C01828=1149.288,-103.464,-43.595,178.756,5.963,149.436
C01829=1149.282,-103.213,-43.605,178.759,5.964,149.436
C01830=1149.276,-102.942,-43.615,178.761,5.964,149.435
C01831=1149.271,-102.669,-43.625,178.763,5.965,149.435
C01832=1149.265,-102.397,-43.635,178.765,5.965,149.434
C01833=1149.260,-102.125,-43.645,178.767,5.965,149.433
C01834=1149.254,-101.875,-43.654,178.770,5.966,149.433
C01835=1149.249,-101.625,-43.664,178.772,5.966,149.432
C01836=1149.243,-101.375,-43.672,178.774,5.967,149.432
C01837=1149.238,-101.125,-43.681,178.775,5.966,149.431
C01838=1149.233,-100.877,-43.691,178.778,5.967,149.431
C01839=1149.227,-100.627,-43.700,178.780,5.968,149.430
C01840=1149.222,-100.377,-43.709,178.782,5.968,149.430
C01841=1149.216,-100.127,-43.718,178.784,5.968,149.429
C01842=1149.211,-99.877,-43.727,178.786,5.969,149.429
C01843=1149.206,-99.628,-43.737,178.788,5.969,149.428
C01844=1149.201,-99.378,-43.746,178.791,5.969,149.427
C01845=1149.195,-99.128,-43.755,178.792,5.969,149.427
C01846=1149.189,-98.878,-43.764,178.794,5.970,149.426
C01847=1149.185,-98.629,-43.774,178.797,5.971,149.426
C01848=1149.179,-98.378,-43.783,178.799,5.970,149.425
C01849=1149.174,-98.129,-43.792,178.801,5.971,149.425
C01850=1149.169,-97.879,-43.802,178.803,5.972,149.424
C01851=1149.163,-97.629,-43.811,178.805,5.972,149.424
C01852=1149.158,-97.379,-43.820,178.807,5.973,149.423
C01853=1149.152,-97.129,-43.829,178.809,5.972,149.423
C01854=1149.147,-96.880,-43.839,178.811,5.973,149.422
C01855=1149.142,-96.630,-43.848,178.813,5.974,149.422
C01856=1149.136,-96.380,-43.858,178.815,5.974,149.421
C01857=1149.131,-96.131,-43.867,178.818,5.974,149.420
C01858=1149.126,-95.881,-43.876,178.820,5.975,149.420
C01859=1149.120,-95.631,-43.886,178.821,5.975,149.419
C01860=1149.115,-95.381,-43.895,178.824,5.976,149.419
C01861=1149.109,-95.131,-43.905,178.826,5.975,149.418
C01862=1149.104,-94.882,-43.914,178.828,5.976,149.418
C01863=1149.099,-94.632,-43.923,178.830,5.977,149.417
C01864=1149.093,-94.382,-43.933,178.832,5.977,149.417
C01865=1149.088,-94.133,-43.942,178.834,5.977,149.416
C01866=1149.082,-93.883,-43.952,178.836,5.978,149.416
C01867=1149.077,-93.633,-43.961,178.838,5.978,149.415
C01868=1149.072,-93.384,-43.970,178.840,5.979,149.415
C01869=1149.066,-93.133,-43.980,178.843,5.979,149.414
C01870=1149.062,-92.884,-43.990,178.845,5.979,149.413
C01871=1149.056,-92.634,-43.999,178.847,5.980,149.413
C01872=1149.051,-92.384,-44.009,178.849,5.980,149.412
C01873=1149.046,-92.134,-44.019,178.851,5.980,149.412
C01874=1149.040,-91.884,-44.027,178.853,5.981,149.411
C01875=1149.035,-91.634,-44.038,178.855,5.982,149.411
C01876=1149.030,-91.385,-44.047,178.857,5.982,149.410
C01877=1149.024,-91.135,-44.057,178.860,5.982,149.410
C01878=1149.019,-90.885,-44.066,178.862,5.983,149.409
C01879=1149.013,-90.636,-44.076,178.863,5.983,149.409
C01880=1149.008,-90.386,-44.085,178.866,5.983,149.408
C01881=1149.003,-90.137,-44.094,178.868,5.984,149.407
C01882=1148.997,-89.886,-44.104,178.870,5.984,149.407
C01883=1148.992,-89.637,-44.113,178.872,5.985,149.406
C01884=1148.987,-89.387,-44.123,178.874,5.984,149.406
C01885=1148.982,-89.137,-44.133,178.876,5.985,149.405
C01886=1148.976,-88.887,-44.142,178.879,5.986,149.405
C01887=1148.971,-88.637,-44.153,178.881,5.986,149.404
C01888=1148.966,-88.388,-44.162,178.883,5.986,149.404
C01889=1148.960,-88.138,-44.172,178.885,5.987,149.403
C01890=1148.955,-87.889,-44.181,178.887,5.987,149.403
C01891=1148.949,-87.639,-44.191,178.889,5.987,149.402
C01892=1148.944,-87.389,-44.200,178.891,5.988,149.401
C01893=1148.939,-87.138,-44.210,178.894,5.989,149.401
C01894=1148.934,-86.889,-44.220,178.895,5.989,149.400
C01895=1148.929,-86.640,-44.230,178.897,5.989,149.400
C01896=1148.923,-86.390,-44.239,178.900,5.990,149.399
C01897=1148.918,-86.140,-44.249,178.902,5.990,149.399
C01898=1148.912,-85.890,-44.259,178.904,5.990,149.398
C01899=1148.907,-85.641,-44.268,178.907,5.991,149.398
C01900=1148.902,-85.391,-44.279,178.908,5.991,149.397
C01901=1148.897,-85.141,-44.288,178.910,5.992,149.397
C01902=1148.891,-84.891,-44.298,178.913,5.992,149.396
C01903=1148.886,-84.642,-44.308,178.915,5.992,149.395
C01904=1148.881,-84.392,-44.317,178.917,5.993,149.395
C01905=1148.875,-84.142,-44.327,178.919,5.993,149.394
C01906=1148.871,-83.892,-44.337,178.921,5.993,149.394
C01907=1148.865,-83.642,-44.347,178.923,5.994,149.393
C01908=1148.859,-83.393,-44.357,178.925,5.995,149.393
C01909=1148.854,-83.143,-44.367,178.928,5.995,149.392
C01910=1148.848,-82.893,-44.376,178.930,5.995,149.392
C01911=1148.844,-82.643,-44.386,178.932,5.996,149.391
C01912=1148.839,-82.394,-44.396,178.934,5.996,149.391
C01913=1148.833,-82.144,-44.406,178.936,5.996,149.390
C01914=1148.828,-81.894,-44.415,178.938,5.997,149.389
C01915=1148.822,-81.645,-44.426,178.941,5.998,149.389
C01916=1148.817,-81.395,-44.436,178.943,5.997,149.388
C01917=1148.812,-81.145,-44.445,178.945,5.998,149.388
C01918=1148.806,-80.895,-44.455,178.947,5.999,149.387
C01919=1148.801,-80.646,-44.466,178.949,5.999,149.387
C01920=1148.796,-80.396,-44.475,178.951,5.999,149.386
C01921=1148.791,-80.146,-44.485,178.954,6.000,149.386
C01922=1148.785,-79.896,-44.495,178.956,6.001,149.385
C01923=1148.779,-79.647,-44.505,178.958,6.000,149.384
C01924=1148.775,-79.397,-44.515,178.960,6.001,149.384
C01925=1148.770,-79.147,-44.526,178.962,6.002,149.383
C01926=1148.764,-78.897,-44.535,178.965,6.002,149.383
C01927=1148.759,-78.648,-44.545,178.966,6.002,149.382
C01928=1148.753,-78.398,-44.555,178.969,6.003,149.382
C01929=1148.748,-78.149,-44.565,178.971,6.003,149.381
C01930=1148.743,-77.898,-44.576,178.973,6.003,149.381
C01931=1148.738,-77.648,-44.585,178.975,6.004,149.380
C01932=1148.732,-77.399,-44.595,178.977,6.005,149.380
C01933=1148.726,-77.149,-44.605,178.980,6.005,149.379
C01934=1148.721,-76.878,-44.616,178.982,6.006,149.378
C01935=1148.715,-76.606,-44.628,178.984,6.005,149.378
C01936=1148.710,-76.335,-44.638,178.986,6.006,149.377
C01937=1148.703,-76.064,-44.649,178.989,6.007,149.377
C01938=1148.698,-75.813,-44.660,178.991,6.007,149.376
C01939=1148.693,-75.564,-44.669,178.993,6.008,149.376
C01940=1148.688,-75.315,-44.679,178.996,6.008,149.375
C01941=1148.682,-75.065,-44.690,178.998,6.008,149.374
C01942=1148.677,-74.815,-44.700,179.000,6.009,149.374
C01943=1148.672,-74.565,-44.710,179.003,6.010,149.373
C01944=1148.667,-74.316,-44.720,179.004,6.010,149.373
C01945=1148.662,-74.066,-44.731,179.006,6.010,149.372
C01946=1148.656,-73.816,-44.741,179.009,6.011,149.372
C01947=1148.650,-73.567,-44.751,179.011,6.012,149.371
C01948=1148.645,-73.317,-44.761,179.013,6.012,149.371
C01949=1148.640,-73.066,-44.771,179.016,6.012,149.370
C01950=1148.634,-72.817,-44.781,179.018,6.013,149.369
C01951=1148.629,-72.568,-44.791,179.020,6.013,149.369
C01952=1148.624,-72.317,-44.801,179.022,6.013,149.368
C01953=1148.619,-72.068,-44.812,179.024,6.014,149.368
C01954=1148.613,-71.818,-44.822,179.026,6.015,149.367
C01955=1148.608,-71.568,-44.832,179.029,6.015,149.366
C01956=1148.602,-71.318,-44.843,179.031,6.015,149.366
C01957=1148.597,-71.069,-44.853,179.033,6.016,149.366
C01958=1148.593,-70.820,-44.863,179.035,6.016,149.365
C01959=1148.587,-70.570,-44.874,179.038,6.017,149.364
C01960=1148.582,-70.321,-44.884,179.039,6.017,149.364
C01961=1148.577,-70.070,-44.894,179.042,6.017,149.363
C01962=1148.571,-69.821,-44.905,179.044,6.018,149.363
C01963=1148.566,-69.570,-44.915,179.046,6.019,149.362
C01964=1148.560,-69.321,-44.925,179.048,6.018,149.361
C01965=1148.555,-69.071,-44.936,179.051,6.019,149.361
C01966=1148.550,-68.821,-44.946,179.053,6.020,149.361
C01967=1148.544,-68.572,-44.956,179.055,6.020,149.360
C01968=1148.539,-68.322,-44.967,179.057,6.020,149.359
C01969=1148.534,-68.072,-44.977,179.059,6.021,149.359
C01970=1148.528,-67.822,-44.987,179.062,6.021,149.358
C01971=1148.524,-67.573,-44.998,179.064,6.022,149.358
C01972=1148.518,-67.323,-45.008,179.066,6.023,149.357
C01973=1148.513,-67.074,-45.019,179.068,6.023,149.356
C01974=1148.508,-66.824,-45.029,179.071,6.023,149.356
C01975=1148.502,-66.574,-45.039,179.073,6.024,149.355
C01976=1148.497,-66.324,-45.050,179.075,6.025,149.355
C01977=1148.492,-66.075,-45.061,179.077,6.024,149.354
C01978=1148.486,-65.825,-45.071,179.080,6.025,149.354
C01979=1148.481,-65.575,-45.082,179.082,6.026,149.353
C01980=1148.476,-65.326,-45.092,179.084,6.026,149.353
C01981=1148.471,-65.075,-45.102,179.087,6.027,149.352
C01982=1148.465,-64.826,-45.113,179.088,6.027,149.351
C01983=1148.460,-64.576,-45.124,179.090,6.028,149.351
C01984=1148.455,-64.327,-45.134,179.093,6.028,149.350
C01985=1148.450,-64.076,-45.145,179.095,6.029,149.350
C01986=1148.444,-63.827,-45.155,179.098,6.030,149.349
C01987=1148.439,-63.578,-45.166,179.100,6.029,149.349
C01988=1148.434,-63.328,-45.176,179.102,6.030,149.348
C01989=1148.428,-63.078,-45.187,179.104,6.031,149.348
C01990=1148.423,-62.828,-45.197,179.107,6.031,149.347
C01991=1148.417,-62.579,-45.209,179.109,6.032,149.346
C01992=1148.412,-62.328,-45.219,179.111,6.031,149.346
C01993=1148.407,-62.079,-45.229,179.113,6.032,149.345
C01994=1148.402,-61.829,-45.241,179.115,6.033,149.345
C01995=1148.396,-61.580,-45.251,179.118,6.033,149.344
C01996=1148.391,-61.329,-45.262,179.120,6.034,149.344
C01997=1148.386,-61.081,-45.272,179.122,6.034,149.343
C01998=1148.381,-60.830,-45.283,179.124,6.035,149.342
C01999=1148.376,-60.581,-45.293,179.127,6.035,149.342
C02000=1148.371,-60.331,-45.305,179.129,6.036,149.341
C02001=1148.365,-60.082,-45.315,179.131,6.036,149.341
C02002=1148.360,-59.831,-45.325,179.133,6.036,149.340
C02003=1148.354,-59.582,-45.337,179.136,6.037,149.340
C02004=1148.349,-59.332,-45.347,179.138,6.038,149.339
C02005=1148.344,-59.082,-45.358,179.140,6.038,149.339
C02006=1148.339,-58.833,-45.369,179.143,6.039,149.338
C02007=1148.333,-58.583,-45.379,179.145,6.040,149.337
C02008=1148.329,-58.334,-45.390,179.147,6.040,149.337
C02009=1148.323,-58.084,-45.401,179.149,6.040,149.336
C02010=1148.318,-57.834,-45.411,179.151,6.041,149.336
C02011=1148.313,-57.584,-45.423,179.154,6.041,149.335
C02012=1148.307,-57.334,-45.433,179.156,6.042,149.335
C02013=1148.302,-57.085,-45.445,179.158,6.042,149.334
C02014=1148.297,-56.835,-45.455,179.161,6.042,149.333
C02015=1148.292,-56.585,-45.466,179.163,6.043,149.333
C02016=1148.287,-56.336,-45.476,179.165,6.044,149.332
C02017=1148.281,-56.085,-45.487,179.168,6.044,149.332
C02018=1148.275,-55.836,-45.498,179.170,6.045,149.331
C02019=1148.270,-55.586,-45.509,179.172,6.045,149.331
C02020=1148.266,-55.337,-45.520,179.174,6.045,149.330
C02021=1148.260,-55.087,-45.530,179.176,6.046,149.330
C02022=1148.255,-54.837,-45.542,179.179,6.047,149.329
C02023=1148.249,-54.588,-45.553,179.181,6.047,149.328
C02024=1148.244,-54.338,-45.564,179.183,6.048,149.328
C02025=1148.240,-54.088,-45.575,179.186,6.049,149.327
C02026=1148.234,-53.839,-45.585,179.188,6.049,149.327
C02027=1148.229,-53.589,-45.597,179.190,6.049,149.326
C02028=1148.223,-53.339,-45.607,179.192,6.050,149.326
C02029=1148.218,-53.090,-45.619,179.195,6.050,149.325
C02030=1148.213,-52.839,-45.629,179.197,6.051,149.324
C02031=1148.207,-52.590,-45.641,179.199,6.052,149.324
C02032=1148.202,-52.340,-45.651,179.202,6.052,149.323
C02033=1148.197,-52.091,-45.662,179.204,6.052,149.323
C02034=1148.192,-51.841,-45.674,179.206,6.053,149.322
C02035=1148.187,-51.591,-45.685,179.209,6.053,149.322
C02036=1148.181,-51.342,-45.696,179.211,6.054,149.321
C02037=1148.176,-51.092,-45.706,179.213,6.055,149.321
C02038=1148.171,-50.821,-45.719,179.216,6.055,149.320
C02039=1148.165,-50.550,-45.730,179.218,6.056,149.319
C02040=1148.159,-50.279,-45.743,179.220,6.056,149.319
C02041=1148.153,-50.009,-45.755,179.223,6.057,149.318
C02042=1148.148,-49.759,-45.766,179.225,6.058,149.318
C02043=1148.143,-49.510,-45.777,179.228,6.058,149.317
C02044=1148.137,-49.260,-45.788,179.230,6.059,149.316
C02045=1148.132,-49.010,-45.799,179.232,6.059,149.316
C02046=1148.128,-48.761,-45.811,179.234,6.059,149.315
C02047=1148.121,-48.511,-45.821,179.237,6.060,149.315
C02048=1148.117,-48.261,-45.833,179.239,6.060,149.314
C02049=1148.112,-48.012,-45.844,179.241,6.061,149.314
C02050=1148.106,-47.762,-45.855,179.244,6.062,149.313
C02051=1148.101,-47.512,-45.866,179.246,6.062,149.312
C02052=1148.095,-47.262,-45.878,179.249,6.063,149.312
C02053=1148.091,-47.013,-45.889,179.251,6.063,149.311
C02054=1148.085,-46.764,-45.900,179.253,6.063,149.311
C02055=1148.080,-46.513,-45.911,179.255,6.064,149.310
C02056=1148.075,-46.263,-45.923,179.258,6.065,149.310
C02057=1148.069,-46.014,-45.934,179.260,6.065,149.309
C02058=1148.064,-45.765,-45.945,179.262,6.066,149.308
C02059=1148.059,-45.514,-45.956,179.265,6.067,149.308
C02060=1148.053,-45.265,-45.967,179.267,6.067,149.307
C02061=1148.049,-45.016,-45.979,179.270,6.068,149.307
C02062=1148.043,-44.766,-45.991,179.271,6.068,149.306
C02063=1148.038,-44.516,-46.002,179.274,6.068,149.305
C02064=1148.032,-44.266,-46.013,179.276,6.069,149.305
C02065=1148.027,-44.016,-46.024,179.278,6.070,149.305
C02066=1148.022,-43.767,-46.036,179.281,6.070,149.304
C02067=1148.017,-43.517,-46.047,179.283,6.071,149.303
C02068=1148.012,-43.268,-46.058,179.286,6.071,149.303
C02069=1148.007,-43.018,-46.070,179.288,6.072,149.302
C02070=1148.002,-42.768,-46.081,179.290,6.073,149.302
C02071=1147.996,-42.518,-46.092,179.293,6.073,149.301
C02072=1147.991,-42.269,-46.103,179.295,6.074,149.301
C02073=1147.985,-42.019,-46.115,179.297,6.074,149.300
C02074=1147.981,-41.769,-46.127,179.299,6.074,149.299
C02075=1147.975,-41.519,-46.138,179.301,6.075,149.299
C02076=1147.970,-41.271,-46.149,179.304,6.076,149.298
C02077=1147.965,-41.021,-46.161,179.306,6.076,149.298
C02078=1147.960,-40.771,-46.173,179.309,6.077,149.297
C02079=1147.955,-40.521,-46.184,179.311,6.078,149.297
C02080=1147.949,-40.271,-46.196,179.314,6.078,149.296
C02081=1147.944,-40.022,-46.207,179.316,6.079,149.295
C02082=1147.938,-39.772,-46.219,179.318,6.080,149.295
C02083=1147.934,-39.523,-46.230,179.321,6.080,149.294
C02084=1147.928,-39.272,-46.242,179.323,6.081,149.294
C02085=1147.923,-39.022,-46.253,179.325,6.080,149.293
C02086=1147.917,-38.773,-46.264,179.327,6.081,149.293
C02087=1147.913,-38.524,-46.276,179.329,6.082,149.292
C02088=1147.907,-38.274,-46.288,179.332,6.082,149.291
C02089=1147.902,-38.024,-46.299,179.334,6.083,149.291
C02090=1147.897,-37.774,-46.311,179.337,6.084,149.290
C02091=1147.892,-37.525,-46.323,179.339,6.084,149.290
C02092=1147.887,-37.276,-46.334,179.341,6.085,149.289
C02093=1147.881,-37.026,-46.346,179.344,6.086,149.289
C02094=1147.876,-36.776,-46.358,179.346,6.086,149.288
C02095=1147.871,-36.526,-46.369,179.349,6.087,149.287
C02096=1147.866,-36.276,-46.381,179.351,6.088,149.287
C02097=1147.860,-36.026,-46.393,179.354,6.088,149.286
C02098=1147.855,-35.778,-46.404,179.356,6.089,149.286
C02099=1147.849,-35.528,-46.416,179.358,6.090,149.285
C02100=1147.844,-35.278,-46.428,179.361,6.090,149.285
C02101=1147.839,-35.028,-46.439,179.363,6.091,149.284
C02102=1147.834,-34.778,-46.451,179.365,6.091,149.283
C02103=1147.829,-34.528,-46.462,179.367,6.091,149.283
C02104=1147.824,-34.279,-46.475,179.370,6.092,149.282
C02105=1147.819,-34.029,-46.487,179.372,6.092,149.282
C02106=1147.813,-33.780,-46.498,179.374,6.093,149.281
C02107=1147.808,-33.530,-46.510,179.377,6.094,149.281
C02108=1147.802,-33.280,-46.521,179.379,6.094,149.280
C02109=1147.797,-33.030,-46.533,179.382,6.095,149.279
C02110=1147.793,-32.781,-46.545,179.384,6.096,149.279
C02111=1147.787,-32.532,-46.557,179.386,6.096,149.278
C02112=1147.782,-32.282,-46.569,179.389,6.097,149.278
C02113=1147.777,-32.032,-46.580,179.391,6.098,149.277
C02114=1147.772,-31.782,-46.592,179.393,6.098,149.277
C02115=1147.767,-31.533,-46.605,179.396,6.099,149.276
C02116=1147.761,-31.283,-46.617,179.398,6.099,149.275
C02117=1147.756,-31.034,-46.628,179.401,6.100,149.275
C02118=1147.750,-30.784,-46.640,179.403,6.101,149.274
C02119=1147.745,-30.535,-46.652,179.405,6.101,149.274
C02120=1147.740,-30.285,-46.664,179.408,6.102,149.273
C02121=1147.735,-30.035,-46.675,179.410,6.102,149.273
C02122=1147.730,-29.785,-46.687,179.412,6.103,149.272
C02123=1147.725,-29.536,-46.700,179.415,6.104,149.271
C02124=1147.719,-29.286,-46.712,179.417,6.104,149.271
C02125=1147.714,-29.036,-46.723,179.419,6.105,149.270
C02126=1147.709,-28.787,-46.736,179.422,6.106,149.270
C02127=1147.704,-28.537,-46.748,179.424,6.106,149.269
C02128=1147.698,-28.287,-46.759,179.427,6.107,149.269
C02129=1147.693,-28.037,-46.771,179.429,6.108,149.268
C02130=1147.689,-27.788,-46.783,179.432,6.108,149.267
C02131=1147.683,-27.538,-46.795,179.434,6.109,149.267
C02132=1147.678,-27.289,-46.808,179.436,6.110,149.266
C02133=1147.673,-27.039,-46.820,179.439,6.110,149.266
C02134=1147.667,-26.789,-46.832,179.441,6.111,149.265
C02135=1147.662,-26.540,-46.844,179.444,6.111,149.265
C02136=1147.657,-26.290,-46.855,179.446,6.112,149.264
C02137=1147.652,-26.040,-46.867,179.448,6.112,149.263
C02138=1147.647,-25.791,-46.880,179.451,6.113,149.263
C02139=1147.641,-25.541,-46.892,179.453,6.114,149.262
C02140=1147.636,-25.292,-46.904,179.456,6.114,149.262
C02141=1147.631,-25.042,-46.916,179.458,6.115,149.261
C02142=1147.626,-24.771,-46.929,179.460,6.116,149.261
C02143=1147.620,-24.502,-46.943,179.463,6.116,149.260
C02144=1147.615,-24.232,-46.956,179.465,6.117,149.259
C02145=1147.609,-23.961,-46.969,179.468,6.118,149.259
C02146=1147.604,-23.712,-46.982,179.471,6.119,149.258
C02147=1147.599,-23.462,-46.993,179.473,6.119,149.258
C02148=1147.594,-23.213,-47.006,179.476,6.120,149.257
C02149=1147.588,-22.963,-47.017,179.478,6.121,149.256
C02150=1147.583,-22.714,-47.030,179.480,6.121,149.256
C02151=1147.578,-22.464,-47.042,179.483,6.122,149.255
C02152=1147.573,-22.214,-47.055,179.485,6.123,149.255
C02153=1147.567,-21.964,-47.066,179.487,6.123,149.254
C02154=1147.562,-21.715,-47.079,179.490,6.124,149.254
C02155=1147.557,-21.465,-47.091,179.492,6.125,149.253
C02156=1147.551,-21.216,-47.104,179.495,6.125,149.252
C02157=1147.546,-20.966,-47.115,179.497,6.126,149.252
C02158=1147.541,-20.717,-47.128,179.499,6.127,149.251
C02159=1147.536,-20.466,-47.140,179.502,6.127,149.251
C02160=1147.531,-20.217,-47.153,179.504,6.128,149.250
C02161=1147.526,-19.967,-47.165,179.507,6.128,149.250
C02162=1147.520,-19.717,-47.177,179.509,6.129,149.249
C02163=1147.515,-19.468,-47.190,179.512,6.129,149.248
C02164=1147.510,-19.218,-47.202,179.514,6.130,149.248
C02165=1147.505,-18.969,-47.214,179.516,6.131,149.247
C02166=1147.500,-18.720,-47.227,179.519,6.131,149.247
C02167=1147.494,-18.470,-47.239,179.521,6.132,149.246
C02168=1147.490,-18.220,-47.252,179.523,6.133,149.246
C02169=1147.485,-17.970,-47.264,179.526,6.133,149.245
C02170=1147.479,-17.720,-47.276,179.528,6.134,149.245
C02171=1147.474,-17.471,-47.289,179.531,6.135,149.244
C02172=1147.469,-17.222,-47.302,179.534,6.136,149.243
C02173=1147.463,-16.972,-47.313,179.536,6.137,149.243
C02174=1147.458,-16.722,-47.326,179.538,6.138,149.242
C02175=1147.453,-16.472,-47.340,179.541,6.138,149.242
C02176=1147.448,-16.222,-47.352,179.543,6.139,149.241
C02177=1147.443,-15.973,-47.364,179.546,6.139,149.241
C02178=1147.437,-15.724,-47.377,179.548,6.140,149.240
C02179=1147.432,-15.474,-47.389,179.550,6.140,149.239
C02180=1147.427,-15.224,-47.401,179.553,6.141,149.239
C02181=1147.422,-14.974,-47.414,179.555,6.142,149.238
C02182=1147.417,-14.725,-47.427,179.557,6.142,149.238
C02183=1147.412,-14.476,-47.439,179.560,6.143,149.237
C02184=1147.407,-14.226,-47.451,179.562,6.144,149.237
C02185=1147.401,-13.976,-47.464,179.564,6.144,149.236
C02186=1147.396,-13.726,-47.477,179.568,6.146,149.235
C02187=1147.391,-13.477,-47.490,179.570,6.146,149.235
C02188=1147.386,-13.227,-47.503,179.573,6.147,149.234
C02189=1147.381,-12.977,-47.515,179.575,6.148,149.234
C02190=1147.375,-12.728,-47.527,179.577,6.148,149.233
C02191=1147.370,-12.478,-47.541,179.580,6.149,149.233
C02192=1147.365,-12.229,-47.553,179.582,6.150,149.232
C02193=1147.360,-11.979,-47.566,179.584,6.150,149.231
C02194=1147.355,-11.730,-47.578,179.587,6.151,149.231
C02195=1147.350,-11.480,-47.591,179.589,6.151,149.230
C02196=1147.345,-11.230,-47.603,179.591,6.152,149.230
C02197=1147.339,-10.980,-47.617,179.595,6.153,149.229
C02198=1147.334,-10.731,-47.629,179.597,6.154,149.229
C02199=1147.329,-10.481,-47.642,179.599,6.155,149.228
C02200=1147.324,-10.232,-47.655,179.602,6.155,149.228
C02201=1147.319,-9.982,-47.667,179.604,6.156,149.227
C02202=1147.313,-9.733,-47.680,179.607,6.157,149.226
C02203=1147.309,-9.483,-47.693,179.609,6.157,149.226
C02204=1147.304,-9.233,-47.706,179.611,6.158,149.225
C02205=1147.298,-8.984,-47.719,179.614,6.159,149.225
C02206=1147.293,-8.734,-47.732,179.616,6.159,149.224
C02207=1147.288,-8.484,-47.745,179.619,6.161,149.224
C02208=1147.283,-8.235,-47.757,179.621,6.162,149.223
C02209=1147.278,-7.986,-47.770,179.624,6.162,149.222
C02210=1147.273,-7.735,-47.784,179.626,6.163,149.222
C02211=1147.267,-7.486,-47.796,179.629,6.163,149.221
C02212=1147.262,-7.237,-47.809,179.631,6.164,149.221
C02213=1147.257,-6.986,-47.822,179.633,6.164,149.220
C02214=1147.252,-6.737,-47.835,179.636,6.165,149.220
C02215=1147.247,-6.488,-47.848,179.638,6.166,149.219
C02216=1147.241,-6.238,-47.861,179.641,6.167,149.218
C02217=1147.236,-5.988,-47.874,179.643,6.168,149.218
C02218=1147.231,-5.739,-47.886,179.646,6.169,149.217
C02219=1147.225,-5.489,-47.899,179.648,6.169,149.217
C02220=1147.221,-5.239,-47.912,179.651,6.170,149.216
C02221=1147.216,-4.990,-47.925,179.653,6.171,149.216
C02222=1147.210,-4.740,-47.938,179.656,6.171,149.215
C02223=1147.205,-4.490,-47.951,179.658,6.173,149.215
C02224=1147.200,-4.241,-47.964,179.661,6.173,149.214
C02225=1147.195,-3.991,-47.978,179.663,6.174,149.213
C02226=1147.190,-3.742,-47.991,179.665,6.175,149.213
C02227=1147.185,-3.493,-48.003,179.668,6.175,149.212
C02228=1147.180,-3.242,-48.017,179.670,6.176,149.212
C02229=1147.175,-2.993,-48.029,179.673,6.176,149.211
C02230=1147.169,-2.743,-48.043,179.676,6.178,149.211
C02231=1147.165,-2.494,-48.056,179.678,6.178,149.210
C02232=1147.160,-2.245,-48.069,179.680,6.179,149.209
C02233=1147.154,-1.994,-48.083,179.683,6.180,149.209
C02234=1147.149,-1.745,-48.095,179.685,6.180,149.208
C02235=1147.143,-1.495,-48.108,179.687,6.181,149.208
C02236=1147.139,-1.246,-48.122,179.690,6.182,149.207
C02237=1147.133,-0.996,-48.135,179.693,6.183,149.207
C02238=1147.128,-0.747,-48.148,179.696,6.184,149.206
C02239=1147.123,-0.497,-48.161,179.698,6.185,149.206
C02240=1147.118,-0.247,-48.174,179.700,6.185,149.205
C02241=1147.113,0.002,-48.188,179.703,6.186,149.204
C02242=1147.108,0.252,-48.201,179.705,6.187,149.204
C02243=1147.103,0.502,-48.214,179.708,6.188,149.203
C02244=1147.098,0.751,-48.228,179.710,6.189,149.203
C02245=1147.092,1.000,-48.240,179.713,6.189,149.202
C02246=1147.087,1.270,-48.255,179.715,6.190,149.202
C02247=1147.081,1.539,-48.270,179.718,6.191,149.201
C02248=1147.075,1.810,-48.284,179.721,6.192,149.200
C02249=1147.070,2.078,-48.298,179.723,6.192,149.200
C02250=1147.065,2.328,-48.311,179.726,6.193,149.199
C02251=1147.060,2.577,-48.325,179.729,6.194,149.199
C02252=1147.055,2.827,-48.338,179.731,6.195,149.198
C02253=1147.050,3.077,-48.351,179.733,6.196,149.197
C02254=1147.045,3.326,-48.365,179.736,6.196,149.197
C02255=1147.040,3.576,-48.378,179.738,6.197,149.196
C02256=1147.034,3.826,-48.391,179.741,6.199,149.196
C02257=1147.029,4.075,-48.405,179.744,6.199,149.195
C02258=1147.024,4.325,-48.418,179.746,6.200,149.195
C02259=1147.019,4.574,-48.432,179.748,6.200,149.194
C02260=1147.014,4.824,-48.445,179.751,6.201,149.194
C02261=1147.008,5.074,-48.458,179.754,6.202,149.193
C02262=1147.003,5.323,-48.473,179.756,6.203,149.192
C02263=1146.998,5.573,-48.485,179.759,6.203,149.192
C02264=1146.993,5.822,-48.499,179.761,6.204,149.191
C02265=1146.988,6.072,-48.512,179.763,6.205,149.191
C02266=1146.983,6.321,-48.526,179.766,6.206,149.190
C02267=1146.977,6.571,-48.540,179.768,6.207,149.190
C02268=1146.973,6.820,-48.553,179.771,6.208,149.189
C02269=1146.967,7.070,-48.566,179.773,6.208,149.188
C02270=1146.963,7.319,-48.580,179.776,6.209,149.188
C02271=1146.957,7.569,-48.593,179.779,6.210,149.187
C02272=1146.952,7.819,-48.608,179.781,6.211,149.187
C02273=1146.947,8.068,-48.620,179.784,6.212,149.186
C02274=1146.942,8.318,-48.634,179.786,6.213,149.186
C02275=1146.937,8.568,-48.648,179.788,6.213,149.185
C02276=1146.932,8.817,-48.661,179.791,6.215,149.185
C02277=1146.927,9.067,-48.676,179.794,6.215,149.184
C02278=1146.921,9.316,-48.689,179.796,6.216,149.183
C02279=1146.916,9.566,-48.703,179.799,6.216,149.183
C02280=1146.911,9.815,-48.716,179.801,6.218,149.182
C02281=1146.906,10.065,-48.730,179.804,6.219,149.182
C02282=1146.901,10.315,-48.744,179.806,6.219,149.181
C02283=1146.896,10.564,-48.757,179.808,6.220,149.181
C02284=1146.891,10.814,-48.771,179.811,6.220,149.180
C02285=1146.885,11.063,-48.784,179.814,6.222,149.180
C02286=1146.880,11.313,-48.799,179.816,6.223,149.179
C02287=1146.876,11.562,-48.812,179.819,6.223,149.178
C02288=1146.870,11.812,-48.825,179.821,6.224,149.178
C02289=1146.865,12.062,-48.840,179.824,6.225,149.177
C02290=1146.860,12.311,-48.854,179.826,6.226,149.177
C02291=1146.856,12.560,-48.867,179.829,6.227,149.176
C02292=1146.850,12.810,-48.881,179.831,6.227,149.176
C02293=1146.845,13.059,-48.895,179.834,6.229,149.175
C02294=1146.840,13.309,-48.909,179.836,6.230,149.174
C02295=1146.835,13.560,-48.923,179.839,6.230,149.174
C02296=1146.830,13.808,-48.936,179.841,6.231,149.173
C02297=1146.825,14.058,-48.950,179.844,6.232,149.173
C02298=1146.820,14.308,-48.965,179.847,6.233,149.172
C02299=1146.814,14.557,-48.978,179.849,6.234,149.172
C02300=1146.809,14.807,-48.992,179.852,6.234,149.171
C02301=1146.804,15.057,-49.006,179.854,6.236,149.171
C02302=1146.799,15.305,-49.020,179.857,6.236,149.170
C02303=1146.794,15.555,-49.034,179.859,6.237,149.169
C02304=1146.789,15.805,-49.047,179.861,6.238,149.169
C02305=1146.784,16.054,-49.061,179.865,6.239,149.168
C02306=1146.779,16.304,-49.076,179.867,6.240,149.168
C02307=1146.774,16.554,-49.090,179.869,6.240,149.167
C02308=1146.768,16.803,-49.104,179.872,6.242,149.167
C02309=1146.763,17.053,-49.118,179.875,6.242,149.166
C02310=1146.759,17.303,-49.131,179.877,6.243,149.166
C02311=1146.753,17.552,-49.145,179.879,6.244,149.165
C02312=1146.748,17.801,-49.159,179.882,6.245,149.164
C02313=1146.743,18.051,-49.174,179.885,6.246,149.164
C02314=1146.738,18.301,-49.188,179.887,6.247,149.163
C02315=1146.733,18.550,-49.202,179.889,6.247,149.163
C02316=1146.728,18.799,-49.216,179.893,6.249,149.162
C02317=1146.723,19.049,-49.230,179.895,6.249,149.162
C02318=1146.718,19.299,-49.245,179.897,6.250,149.161
C02319=1146.712,19.548,-49.258,179.900,6.252,149.161
C02320=1146.707,19.798,-49.273,179.902,6.252,149.160
C02321=1146.702,20.047,-49.287,179.905,6.253,149.159
C02322=1146.697,20.298,-49.301,179.908,6.254,149.159
C02323=1146.691,20.547,-49.314,179.910,6.255,149.158
C02324=1146.686,20.796,-49.329,179.913,6.256,149.158
C02325=1146.682,21.046,-49.343,179.915,6.257,149.157
C02326=1146.677,21.296,-49.357,179.918,6.258,149.157
C02327=1146.671,21.545,-49.371,179.920,6.259,149.156
C02328=1146.666,21.794,-49.386,179.923,6.259,149.156
C02329=1146.661,22.044,-49.400,179.926,6.261,149.155
C02330=1146.656,22.293,-49.415,179.928,6.261,149.154
C02331=1146.652,22.543,-49.429,179.930,6.262,149.154
C02332=1146.646,22.792,-49.443,179.933,6.264,149.154
C02333=1146.641,23.042,-49.457,179.936,6.264,149.153
C02334=1146.636,23.291,-49.471,179.938,6.265,149.152
C02335=1146.631,23.541,-49.486,179.941,6.265,149.152
C02336=1146.626,23.791,-49.500,179.943,6.267,149.151
C02337=1146.621,24.040,-49.514,179.946,6.267,149.151
C02338=1146.616,24.290,-49.528,179.948,6.268,149.150
C02339=1146.611,24.539,-49.543,179.951,6.270,149.150
C02340=1146.606,24.788,-49.558,179.954,6.270,149.149
C02341=1146.601,25.038,-49.572,179.956,6.271,149.149
C02342=1146.596,25.288,-49.586,179.959,6.272,149.148
C02343=1146.591,25.537,-49.600,179.961,6.273,149.147
C02344=1146.585,25.787,-49.615,179.963,6.274,149.147
C02345=1146.580,26.037,-49.629,179.967,6.275,149.146
C02346=1146.575,26.286,-49.644,179.969,6.276,149.146
C02347=1146.570,26.535,-49.658,179.971,6.277,149.145
C02348=1146.565,26.785,-49.673,179.974,6.278,149.145
C02349=1146.560,27.035,-49.687,179.977,6.279,149.144
C02350=1146.555,27.303,-49.702,179.980,6.280,149.144
C02351=1146.549,27.572,-49.719,179.982,6.281,149.143
C02352=1146.543,27.841,-49.734,179.985,6.282,149.142
C02353=1146.538,28.110,-49.749,179.988,6.283,149.142
C02354=1146.533,28.360,-49.764,179.990,6.284,149.141
C02355=1146.528,28.609,-49.779,179.993,6.285,149.141
C02356=1146.523,28.859,-49.793,179.995,6.286,149.140
C02357=1146.518,29.109,-49.808,179.998,6.287,149.139
C02358=1146.513,29.358,-49.822,-179.999,6.288,149.139
C02359=1146.508,29.608,-49.837,-179.997,6.288,149.138
C02360=1146.502,29.857,-49.851,-179.994,6.290,149.138
C02361=1146.497,30.107,-49.866,-179.992,6.291,149.137
C02362=1146.492,30.356,-49.881,-179.989,6.291,149.137
C02363=1146.488,30.605,-49.895,-179.986,6.293,149.136
C02364=1146.482,30.855,-49.910,-179.984,6.293,149.136
C02365=1146.477,31.104,-49.925,-179.982,6.294,149.135
C02366=1146.472,31.354,-49.939,-179.979,6.296,149.135
C02367=1146.468,31.603,-49.954,-179.976,6.296,149.134
C02368=1146.462,31.853,-49.969,-179.973,6.298,149.134
C02369=1146.457,32.103,-49.983,-179.971,6.298,149.133
C02370=1146.452,32.352,-49.998,-179.969,6.299,149.132
C02371=1146.447,32.602,-50.013,-179.966,6.301,149.132
C02372=1146.442,32.851,-50.028,-179.963,6.301,149.131
C02373=1146.437,33.101,-50.042,-179.961,6.302,149.131
C02374=1146.432,33.350,-50.057,-179.958,6.303,149.130
C02375=1146.427,33.600,-50.072,-179.956,6.304,149.130
C02376=1146.422,33.850,-50.087,-179.952,6.305,149.129
C02377=1146.417,34.099,-50.102,-179.950,6.306,149.129
C02378=1146.411,34.349,-50.116,-179.948,6.307,149.128
C02379=1146.407,34.598,-50.131,-179.945,6.308,149.127
C02380=1146.402,34.848,-50.146,-179.943,6.309,149.127
C02381=1146.396,35.097,-50.161,-179.939,6.310,149.126
C02382=1146.391,35.347,-50.176,-179.937,6.311,149.126
C02383=1146.387,35.596,-50.191,-179.935,6.312,149.125
C02384=1146.381,35.845,-50.206,-179.932,6.313,149.125
C02385=1146.376,36.095,-50.220,-179.930,6.314,149.124
C02386=1146.372,36.344,-50.235,-179.926,6.315,149.124
C02387=1146.366,36.594,-50.250,-179.924,6.316,149.123
C02388=1146.361,36.843,-50.265,-179.922,6.317,149.123
C02389=1146.356,37.093,-50.280,-179.919,6.318,149.122
C02390=1146.351,37.342,-50.295,-179.917,6.319,149.122
C02391=1146.346,37.591,-50.310,-179.913,6.321,149.121
C02392=1146.341,37.841,-50.325,-179.911,6.321,149.121
C02393=1146.336,38.090,-50.340,-179.909,6.322,149.120
C02394=1146.330,38.341,-50.355,-179.906,6.323,149.119
C02395=1146.326,38.590,-50.370,-179.904,6.324,149.119
C02396=1146.320,38.839,-50.385,-179.900,6.326,149.118
C02397=1146.315,39.089,-50.400,-179.898,6.326,149.118
C02398=1146.310,39.338,-50.415,-179.896,6.327,149.117
C02399=1146.306,39.588,-50.431,-179.893,6.329,149.117
C02400=1146.300,39.838,-50.446,-179.891,6.329,149.116
C02401=1146.296,40.087,-50.461,-179.888,6.331,149.116
C02402=1146.290,40.336,-50.476,-179.885,6.331,149.115
C02403=1146.286,40.586,-50.491,-179.883,6.333,149.115
C02404=1146.280,40.836,-50.506,-179.880,6.334,149.114
C02405=1146.275,41.085,-50.521,-179.878,6.334,149.114
C02406=1146.270,41.334,-50.537,-179.875,6.336,149.113
C02407=1146.265,41.583,-50.552,-179.872,6.336,149.112
C02408=1146.260,41.833,-50.566,-179.870,6.338,149.112
C02409=1146.255,42.083,-50.582,-179.867,6.339,149.111
C02410=1146.250,42.332,-50.597,-179.864,6.340,149.111
C02411=1146.245,42.581,-50.612,-179.862,6.341,149.110
C02412=1146.240,42.831,-50.627,-179.859,6.342,149.110
C02413=1146.235,43.081,-50.642,-179.857,6.343,149.109
C02414=1146.230,43.330,-50.658,-179.854,6.344,149.109
C02415=1146.225,43.579,-50.673,-179.851,6.345,149.108
C02416=1146.220,43.829,-50.689,-179.849,6.346,149.108
C02417=1146.215,44.079,-50.704,-179.846,6.347,149.107
C02418=1146.210,44.328,-50.719,-179.844,6.348,149.107
C02419=1146.205,44.578,-50.734,-179.840,6.350,149.106
C02420=1146.200,44.827,-50.749,-179.838,6.350,149.106
C02421=1146.195,45.076,-50.765,-179.836,6.352,149.105
C02422=1146.190,45.326,-50.781,-179.833,6.352,149.104
C02423=1146.185,45.575,-50.796,-179.830,6.354,149.104
C02424=1146.180,45.825,-50.811,-179.828,6.355,149.103
C02425=1146.175,46.074,-50.826,-179.825,6.356,149.103
C02426=1146.170,46.323,-50.842,-179.823,6.357,149.102
C02427=1146.165,46.573,-50.858,-179.820,6.358,149.102
C02428=1146.160,46.822,-50.873,-179.817,6.359,149.101
C02429=1146.155,47.072,-50.888,-179.815,6.360,149.101
C02430=1146.149,47.321,-50.904,-179.812,6.361,149.100
C02431=1146.145,47.571,-50.919,-179.810,6.362,149.100
C02432=1146.140,47.820,-50.935,-179.807,6.364,149.099
C02433=1146.135,48.070,-50.951,-179.804,6.364,149.099
C02434=1146.130,48.319,-50.966,-179.802,6.366,149.098
C02435=1146.125,48.569,-50.982,-179.799,6.366,149.097
C02436=1146.120,48.818,-50.997,-179.796,6.368,149.097
C02437=1146.114,49.068,-51.013,-179.794,6.369,149.097
C02438=1146.110,49.317,-51.028,-179.791,6.370,149.096
C02439=1146.105,49.567,-51.044,-179.789,6.371,149.095
C02440=1146.100,49.816,-51.059,-179.786,6.373,149.095
C02441=1146.094,50.066,-51.075,-179.783,6.373,149.094
C02442=1146.090,50.315,-51.090,-179.780,6.375,149.094
C02443=1146.085,50.565,-51.106,-179.778,6.375,149.093
C02444=1146.079,50.814,-51.121,-179.775,6.377,149.093
C02445=1146.074,51.064,-51.137,-179.773,6.378,149.092
C02446=1146.070,51.314,-51.152,-179.770,6.379,149.092
C02447=1146.065,51.562,-51.169,-179.767,6.380,149.091
C02448=1146.059,51.812,-51.184,-179.765,6.381,149.091
C02449=1146.054,52.061,-51.200,-179.762,6.382,149.090
C02450=1146.050,52.311,-51.215,-179.759,6.384,149.090
C02451=1146.045,52.560,-51.231,-179.757,6.384,149.089
C02452=1146.039,52.810,-51.246,-179.754,6.386,149.089
C02453=1146.035,53.059,-51.263,-179.752,6.387,149.088
C02454=1146.029,53.328,-51.280,-179.749,6.388,149.087
C02455=1146.023,53.597,-51.296,-179.746,6.389,149.087
C02456=1146.018,53.865,-51.313,-179.743,6.391,149.086
C02457=1146.012,54.134,-51.330,-179.740,6.392,149.086
C02458=1146.009,54.383,-51.346,-179.737,6.393,149.085
C02459=1146.003,54.632,-51.362,-179.735,6.394,149.085
C02460=1145.998,54.883,-51.378,-179.732,6.395,149.084
C02461=1145.993,55.132,-51.394,-179.730,6.396,149.084
C02462=1145.988,55.381,-51.410,-179.727,6.397,149.083
C02463=1145.983,55.631,-51.426,-179.724,6.398,149.083
C02464=1145.978,55.880,-51.441,-179.721,6.400,149.082
C02465=1145.973,56.129,-51.458,-179.719,6.400,149.082
C02466=1145.968,56.379,-51.474,-179.716,6.402,149.081
C02467=1145.962,56.629,-51.489,-179.713,6.403,149.081
C02468=1145.958,56.877,-51.505,-179.711,6.404,149.080
C02469=1145.953,57.127,-51.521,-179.708,6.406,149.080
C02470=1145.948,57.376,-51.537,-179.706,6.406,149.079
C02471=1145.943,57.626,-51.553,-179.703,6.408,149.079
C02472=1145.938,57.875,-51.569,-179.700,6.409,149.078
C02473=1145.933,58.125,-51.584,-179.698,6.410,149.078
C02474=1145.928,58.374,-51.601,-179.695,6.411,149.077
C02475=1145.923,58.624,-51.617,-179.692,6.412,149.076
C02476=1145.918,58.873,-51.633,-179.690,6.414,149.076
C02477=1145.913,59.123,-51.649,-179.687,6.415,149.076
C02478=1145.908,59.372,-51.666,-179.684,6.416,149.075
C02479=1145.903,59.621,-51.681,-179.682,6.417,149.074
C02480=1145.899,59.871,-51.698,-179.679,6.418,149.074
C02481=1145.893,60.120,-51.713,-179.677,6.419,149.073
C02482=1145.888,60.370,-51.729,-179.674,6.421,149.073
C02483=1145.883,60.619,-51.746,-179.671,6.421,149.072
C02484=1145.878,60.869,-51.761,-179.668,6.423,149.072
C02485=1145.873,61.118,-51.778,-179.666,6.424,149.071
C02486=1145.868,61.367,-51.793,-179.663,6.425,149.071
C02487=1145.864,61.617,-51.810,-179.660,6.427,149.070
C02488=1145.859,61.866,-51.826,-179.658,6.427,149.070
C02489=1145.853,62.116,-51.843,-179.655,6.429,149.069
C02490=1145.848,62.365,-51.859,-179.652,6.430,149.069
C02491=1145.843,62.615,-51.875,-179.650,6.431,149.068
C02492=1145.838,62.864,-51.892,-179.647,6.433,149.068
C02493=1145.833,63.114,-51.908,-179.645,6.433,149.067
C02494=1145.828,63.363,-51.924,-179.642,6.435,149.067
C02495=1145.824,63.612,-51.941,-179.639,6.436,149.066
C02496=1145.818,63.862,-51.956,-179.637,6.437,149.066
C02497=1145.814,64.111,-51.973,-179.634,6.439,149.065
C02498=1145.808,64.360,-51.988,-179.631,6.439,149.065
C02499=1145.803,64.610,-52.006,-179.628,6.441,149.064
C02500=1145.798,64.859,-52.022,-179.626,6.442,149.064
C02501=1145.793,65.109,-52.038,-179.623,6.443,149.063
C02502=1145.789,65.359,-52.055,-179.620,6.445,149.063
C02503=1145.784,65.607,-52.071,-179.618,6.446,149.062
C02504=1145.779,65.857,-52.088,-179.615,6.447,149.062
C02505=1145.773,66.107,-52.104,-179.613,6.448,149.061
C02506=1145.769,66.356,-52.120,-179.610,6.449,149.061
C02507=1145.764,66.605,-52.137,-179.607,6.451,149.060
C02508=1145.759,66.855,-52.153,-179.605,6.452,149.060
C02509=1145.754,67.104,-52.169,-179.602,6.453,149.059
C02510=1145.749,67.353,-52.186,-179.599,6.455,149.059
C02511=1145.744,67.603,-52.203,-179.596,6.455,149.058
C02512=1145.739,67.852,-52.219,-179.594,6.457,149.058
C02513=1145.734,68.102,-52.235,-179.592,6.458,149.057
C02514=1145.729,68.351,-52.251,-179.588,6.459,149.056
C02515=1145.724,68.601,-52.269,-179.586,6.461,149.056
C02516=1145.719,68.850,-52.285,-179.583,6.462,149.056
C02517=1145.714,69.099,-52.302,-179.580,6.463,149.055
C02518=1145.710,69.349,-52.318,-179.577,6.465,149.055
C02519=1145.704,69.599,-52.335,-179.575,6.466,149.054
C02520=1145.699,69.847,-52.351,-179.572,6.467,149.053
C02521=1145.695,70.097,-52.368,-179.570,6.468,149.053
C02522=1145.689,70.346,-52.385,-179.567,6.469,149.053
C02523=1145.684,70.596,-52.401,-179.564,6.471,149.052
C02524=1145.680,70.845,-52.418,-179.562,6.471,149.051
C02525=1145.674,71.094,-52.435,-179.559,6.473,149.051
C02526=1145.669,71.344,-52.451,-179.556,6.475,149.051
C02527=1145.665,71.594,-52.468,-179.554,6.475,149.050
C02528=1145.659,71.843,-52.484,-179.551,6.477,149.050
C02529=1145.655,72.092,-52.501,-179.548,6.479,149.049
C02530=1145.650,72.342,-52.518,-179.546,6.479,149.048
C02531=1145.644,72.591,-52.535,-179.543,6.481,149.048
C02532=1145.640,72.840,-52.551,-179.540,6.482,149.048
C02533=1145.635,73.090,-52.568,-179.537,6.483,149.047
C02534=1145.630,73.339,-52.585,-179.535,6.485,149.046
C02535=1145.625,73.588,-52.602,-179.532,6.486,149.046
C02536=1145.621,73.838,-52.618,-179.530,6.487,149.046
C02537=1145.615,74.088,-52.636,-179.527,6.488,149.045
C02538=1145.610,74.336,-52.652,-179.524,6.490,149.045
C02539=1145.605,74.586,-52.669,-179.522,6.491,149.044
C02540=1145.601,74.836,-52.686,-179.518,6.492,149.043
C02541=1145.595,75.085,-52.703,-179.516,6.494,149.043
C02542=1145.591,75.334,-52.720,-179.514,6.495,149.043
C02543=1145.586,75.583,-52.737,-179.511,6.496,149.042
C02544=1145.581,75.833,-52.754,-179.508,6.498,149.042
C02545=1145.576,76.082,-52.770,-179.505,6.499,149.041
C02546=1145.571,76.332,-52.788,-179.503,6.500,149.041
C02547=1145.566,76.581,-52.804,-179.500,6.502,149.040
C02548=1145.561,76.831,-52.822,-179.497,6.502,149.040
C02549=1145.556,77.080,-52.838,-179.495,6.504,149.039
C02550=1145.551,77.329,-52.856,-179.492,6.506,149.039
C02551=1145.546,77.578,-52.872,-179.489,6.506,149.038
C02552=1145.541,77.828,-52.890,-179.487,6.508,149.038
C02553=1145.536,78.077,-52.906,-179.484,6.510,149.037
C02554=1145.531,78.327,-52.923,-179.481,6.511,149.037
C02555=1145.526,78.576,-52.940,-179.478,6.512,149.036
C02556=1145.522,78.825,-52.958,-179.476,6.513,149.036
C02557=1145.517,79.075,-52.975,-179.473,6.515,149.035
C02558=1145.511,79.343,-52.993,-179.470,6.516,149.035
C02559=1145.506,79.612,-53.012,-179.468,6.517,149.034
C02560=1145.500,79.880,-53.029,-179.464,6.518,149.034
C02561=1145.495,80.149,-53.048,-179.462,6.520,149.033
C02562=1145.490,80.398,-53.066,-179.459,6.522,149.033
C02563=1145.486,80.647,-53.083,-179.456,6.523,149.032
C02564=1145.480,80.897,-53.100,-179.453,6.524,149.032
C02565=1145.476,81.145,-53.117,-179.451,6.526,149.031
C02566=1145.470,81.395,-53.134,-179.448,6.527,149.031
C02567=1145.465,81.645,-53.152,-179.445,6.529,149.030
C02568=1145.461,81.894,-53.169,-179.443,6.529,149.030
C02569=1145.456,82.143,-53.186,-179.440,6.531,149.029
C02570=1145.451,82.393,-53.203,-179.437,6.532,149.029
C02571=1145.446,82.641,-53.220,-179.434,6.534,149.028
C02572=1145.441,82.891,-53.238,-179.432,6.535,149.028
C02573=1145.436,83.140,-53.255,-179.429,6.537,149.027
C02574=1145.431,83.390,-53.272,-179.426,6.538,149.027
C02575=1145.426,83.640,-53.290,-179.424,6.539,149.026
C02576=1145.422,83.889,-53.307,-179.421,6.541,149.026
C02577=1145.417,84.138,-53.324,-179.418,6.542,149.025
C02578=1145.412,84.388,-53.342,-179.415,6.543,149.025
C02579=1145.407,84.637,-53.359,-179.413,6.544,149.024
C02580=1145.402,84.885,-53.377,-179.410,6.546,149.024
C02581=1145.396,85.135,-53.394,-179.407,6.548,149.023
C02582=1145.392,85.384,-53.412,-179.404,6.549,149.023
C02583=1145.387,85.634,-53.428,-179.402,6.550,149.022
C02584=1145.382,85.883,-53.446,-179.399,6.552,149.022
C02585=1145.377,86.133,-53.464,-179.396,6.553,149.022
C02586=1145.372,86.382,-53.482,-179.393,6.555,149.021
C02587=1145.368,86.632,-53.498,-179.391,6.555,149.020
C02588=1145.363,86.881,-53.516,-179.388,6.557,149.020
C02589=1145.357,87.131,-53.534,-179.386,6.559,149.020
C02590=1145.353,87.380,-53.552,-179.382,6.560,149.019
C02591=1145.348,87.629,-53.568,-179.380,6.561,149.019
C02592=1145.343,87.878,-53.586,-179.378,6.563,149.018
C02593=1145.338,88.128,-53.604,-179.375,6.564,149.018
C02594=1145.333,88.377,-53.621,-179.372,6.566,149.017
C02595=1145.328,88.627,-53.639,-179.369,6.567,149.017
C02596=1145.324,88.875,-53.657,-179.367,6.568,149.016
C02597=1145.319,89.125,-53.674,-179.364,6.570,149.016
C02598=1145.314,89.374,-53.692,-179.361,6.571,149.015
C02599=1145.309,89.624,-53.710,-179.358,6.573,149.015
C02600=1145.304,89.873,-53.727,-179.356,6.574,149.014
C02601=1145.299,90.122,-53.745,-179.353,6.575,149.014
C02602=1145.294,90.372,-53.763,-179.350,6.577,149.013
C02603=1145.289,90.621,-53.780,-179.347,6.578,149.013
C02604=1145.284,90.870,-53.798,-179.344,6.580,149.012
C02605=1145.280,91.119,-53.816,-179.342,6.581,149.012
C02606=1145.275,91.369,-53.834,-179.340,6.583,149.012
C02607=1145.269,91.618,-53.851,-179.337,6.584,149.011
C02608=1145.264,91.868,-53.869,-179.334,6.585,149.010
C02609=1145.260,92.117,-53.887,-179.331,6.587,149.010
C02610=1145.255,92.366,-53.905,-179.329,6.588,149.010
C02611=1145.249,92.616,-53.922,-179.326,6.590,149.009
C02612=1145.245,92.865,-53.940,-179.323,6.591,149.009
C02613=1145.240,93.114,-53.958,-179.320,6.593,149.008
C02614=1145.235,93.363,-53.976,-179.317,6.594,149.008
C02615=1145.231,93.612,-53.994,-179.315,6.595,149.007
C02616=1145.226,93.861,-54.012,-179.312,6.597,149.007
C02617=1145.220,94.111,-54.029,-179.309,6.598,149.006
C02618=1145.215,94.360,-54.047,-179.306,6.600,149.006
C02619=1145.211,94.609,-54.065,-179.304,6.602,149.005
C02620=1145.206,94.859,-54.083,-179.302,6.602,149.005
C02621=1145.201,95.109,-54.101,-179.299,6.604,149.005
C02622=1145.196,95.358,-54.119,-179.296,6.605,149.004
C02623=1145.192,95.607,-54.137,-179.293,6.607,149.004
C02624=1145.187,95.856,-54.155,-179.290,6.609,149.003
C02625=1145.182,96.105,-54.173,-179.287,6.610,149.003
C02626=1145.177,96.354,-54.191,-179.285,6.611,149.002
C02627=1145.171,96.604,-54.210,-179.282,6.613,149.002
C02628=1145.166,96.853,-54.228,-179.279,6.614,149.001
C02629=1145.162,97.104,-54.245,-179.277,6.616,149.001
C02630=1145.157,97.353,-54.263,-179.274,6.618,149.000
C02631=1145.152,97.602,-54.281,-179.271,6.619,149.000
C02632=1145.147,97.850,-54.300,-179.269,6.620,148.999
C02633=1145.142,98.100,-54.318,-179.266,6.622,148.999
C02634=1145.137,98.349,-54.336,-179.263,6.623,148.998
C02635=1145.133,98.599,-54.354,-179.260,6.625,148.998
C02636=1145.128,98.848,-54.372,-179.258,6.627,148.998
C02637=1145.123,99.097,-54.390,-179.255,6.628,148.997
C02638=1145.118,99.346,-54.408,-179.252,6.630,148.997
C02639=1145.113,99.596,-54.427,-179.250,6.630,148.996
C02640=1145.108,99.845,-54.445,-179.247,6.632,148.996
C02641=1145.103,100.095,-54.463,-179.244,6.634,148.995
C02642=1145.099,100.344,-54.481,-179.241,6.636,148.995
C02643=1145.094,100.593,-54.499,-179.238,6.637,148.994
C02644=1145.089,100.842,-54.518,-179.235,6.639,148.994
C02645=1145.083,101.091,-54.536,-179.233,6.640,148.993
C02646=1145.079,101.341,-54.555,-179.231,6.641,148.993
C02647=1145.074,101.590,-54.573,-179.228,6.643,148.993
C02648=1145.069,101.839,-54.591,-179.225,6.644,148.992
C02649=1145.064,102.089,-54.609,-179.222,6.646,148.992
C02650=1145.060,102.338,-54.628,-179.219,6.647,148.991
C02651=1145.055,102.587,-54.646,-179.216,6.649,148.991
C02652=1145.050,102.837,-54.664,-179.214,6.651,148.990
C02653=1145.045,103.086,-54.682,-179.211,6.653,148.990
C02654=1145.040,103.335,-54.702,-179.209,6.653,148.989
C02655=1145.035,103.584,-54.720,-179.206,6.655,148.989
C02656=1145.030,103.834,-54.738,-179.203,6.656,148.988
C02657=1145.025,104.083,-54.756,-179.200,6.658,148.988
C02658=1145.021,104.332,-54.775,-179.197,6.660,148.988
C02659=1145.016,104.582,-54.793,-179.195,6.661,148.987
C02660=1145.011,104.831,-54.811,-179.192,6.663,148.987
C02661=1145.006,105.079,-54.830,-179.189,6.664,148.986
C02662=1145.001,105.349,-54.851,-179.186,6.666,148.986
C02663=1144.996,105.617,-54.870,-179.183,6.668,148.985
C02664=1144.990,105.885,-54.890,-179.181,6.670,148.985
C02665=1144.985,106.153,-54.910,-179.177,6.671,148.984
C02666=1144.980,106.403,-54.929,-179.175,6.673,148.984
C02667=1144.975,106.652,-54.947,-179.172,6.674,148.983
C02668=1144.971,106.901,-54.966,-179.169,6.676,148.983
C02669=1144.966,107.151,-54.985,-179.166,6.678,148.983
C02670=1144.961,107.400,-55.003,-179.163,6.679,148.982
C02671=1144.956,107.649,-55.021,-179.160,6.681,148.982
C02672=1144.951,107.898,-55.041,-179.158,6.682,148.981
C02673=1144.947,108.148,-55.059,-179.156,6.683,148.981
C02674=1144.941,108.396,-55.078,-179.153,6.685,148.980
C02675=1144.937,108.646,-55.097,-179.150,6.687,148.980
C02676=1144.932,108.895,-55.115,-179.147,6.688,148.980
C02677=1144.927,109.144,-55.134,-179.145,6.690,148.979
C02678=1144.922,109.394,-55.152,-179.141,6.691,148.979
C02679=1144.917,109.643,-55.171,-179.139,6.693,148.978
C02680=1144.913,109.892,-55.191,-179.136,6.695,148.978
C02681=1144.907,110.142,-55.209,-179.133,6.696,148.977
C02682=1144.903,110.390,-55.228,-179.131,6.698,148.977
C02683=1144.898,110.640,-55.246,-179.128,6.700,148.976
C02684=1144.893,110.889,-55.265,-179.125,6.701,148.976
C02685=1144.889,111.139,-55.284,-179.122,6.703,148.976
C02686=1144.883,111.388,-55.303,-179.119,6.704,148.975
C02687=1144.879,111.636,-55.322,-179.116,6.706,148.975
C02688=1144.874,111.887,-55.341,-179.114,6.708,148.974
C02689=1144.869,112.135,-55.359,-179.112,6.709,148.974
C02690=1144.864,112.385,-55.378,-179.109,6.710,148.973
C02691=1144.859,112.634,-55.397,-179.106,6.712,148.973
C02692=1144.854,112.883,-55.416,-179.103,6.714,148.973
C02693=1144.849,113.133,-55.435,-179.101,6.715,148.972
C02694=1144.844,113.382,-55.454,-179.098,6.717,148.972
C02695=1144.840,113.631,-55.474,-179.095,6.718,148.971
C02696=1144.835,113.880,-55.492,-179.092,6.720,148.971
C02697=1144.830,114.130,-55.511,-179.089,6.722,148.970
C02698=1144.825,114.378,-55.530,-179.087,6.723,148.970
C02699=1144.821,114.628,-55.550,-179.084,6.725,148.970
C02700=1144.815,114.877,-55.569,-179.081,6.727,148.969
C02701=1144.811,115.127,-55.587,-179.078,6.729,148.969
C02702=1144.806,115.376,-55.607,-179.076,6.730,148.968
C02703=1144.802,115.625,-55.626,-179.073,6.732,148.968
C02704=1144.796,115.874,-55.645,-179.070,6.734,148.967
C02705=1144.791,116.124,-55.664,-179.067,6.735,148.967
C02706=1144.787,116.372,-55.683,-179.064,6.737,148.966
C02707=1144.782,116.622,-55.702,-179.062,6.738,148.966
C02708=1144.777,116.871,-55.721,-179.059,6.740,148.966
C02709=1144.773,117.120,-55.741,-179.056,6.742,148.965
C02710=1144.767,117.369,-55.760,-179.053,6.743,148.965
C02711=1144.763,117.618,-55.779,-179.051,6.745,148.964
C02712=1144.758,117.868,-55.797,-179.048,6.747,148.964
C02713=1144.753,118.117,-55.817,-179.045,6.749,148.964
C02714=1144.748,118.366,-55.836,-179.042,6.750,148.963
C02715=1144.744,118.615,-55.855,-179.040,6.752,148.963
C02716=1144.738,118.864,-55.875,-179.037,6.754,148.962
C02717=1144.733,119.114,-55.894,-179.034,6.755,148.962
C02718=1144.729,119.363,-55.913,-179.031,6.757,148.961
C02719=1144.724,119.612,-55.933,-179.028,6.758,148.961
C02720=1144.719,119.862,-55.952,-179.026,6.760,148.961
C02721=1144.714,120.110,-55.972,-179.023,6.762,148.960
C02722=1144.710,120.360,-55.991,-179.020,6.763,148.960
C02723=1144.705,120.609,-56.010,-179.017,6.765,148.959
C02724=1144.700,120.858,-56.030,-179.015,6.767,148.959
C02725=1144.695,121.108,-56.049,-179.012,6.769,148.959
C02726=1144.691,121.356,-56.068,-179.009,6.770,148.958
C02727=1144.686,121.606,-56.088,-179.007,6.772,148.958
C02728=1144.680,121.855,-56.107,-179.004,6.774,148.957
C02729=1144.676,122.104,-56.127,-179.001,6.775,148.957
C02730=1144.671,122.354,-56.146,-178.998,6.777,148.957
C02731=1144.666,122.602,-56.165,-178.996,6.779,148.956
C02732=1144.662,122.852,-56.185,-178.993,6.780,148.956
C02733=1144.657,123.101,-56.205,-178.990,6.782,148.955
C02734=1144.652,123.350,-56.224,-178.987,6.783,148.955
C02735=1144.647,123.599,-56.244,-178.984,6.785,148.954
C02736=1144.642,123.849,-56.264,-178.982,6.787,148.954
C02737=1144.637,124.098,-56.283,-178.979,6.789,148.954
C02738=1144.633,124.347,-56.302,-178.976,6.790,148.953
C02739=1144.629,124.596,-56.322,-178.973,6.792,148.953
C02740=1144.623,124.845,-56.342,-178.971,6.794,148.952
C02741=1144.618,125.094,-56.361,-178.968,6.795,148.952
C02742=1144.614,125.344,-56.381,-178.965,6.797,148.952
C02743=1144.608,125.593,-56.400,-178.962,6.800,148.951
C02744=1144.604,125.842,-56.421,-178.959,6.801,148.951
C02745=1144.599,126.091,-56.440,-178.957,6.803,148.950
C02746=1144.594,126.340,-56.460,-178.954,6.805,148.950
C02747=1144.589,126.590,-56.479,-178.951,6.806,148.950
C02748=1144.585,126.838,-56.499,-178.948,6.808,148.949
C02749=1144.581,127.088,-56.519,-178.946,6.810,148.949
C02750=1144.575,127.337,-56.538,-178.943,6.811,148.948
C02751=1144.571,127.586,-56.558,-178.940,6.813,148.948
C02752=1144.566,127.835,-56.578,-178.937,6.815,148.948
C02753=1144.561,128.085,-56.598,-178.935,6.816,148.947
C02754=1144.556,128.333,-56.618,-178.932,6.818,148.947
C02755=1144.552,128.583,-56.637,-178.929,6.820,148.946
C02756=1144.547,128.832,-56.657,-178.927,6.822,148.946
C02757=1144.542,129.081,-56.677,-178.924,6.823,148.946
C02758=1144.537,129.330,-56.697,-178.921,6.826,148.945
C02759=1144.533,129.579,-56.717,-178.918,6.828,148.945
C02760=1144.528,129.829,-56.737,-178.915,6.829,148.944
C02761=1144.522,130.079,-56.757,-178.912,6.831,148.944
C02762=1144.517,130.327,-56.777,-178.910,6.833,148.944
C02763=1144.513,130.576,-56.797,-178.907,6.834,148.943
C02764=1144.508,130.825,-56.817,-178.904,6.836,148.943
C02765=1144.504,131.075,-56.837,-178.902,6.838,148.942
C02766=1144.499,131.343,-56.858,-178.898,6.840,148.942
C02767=1144.493,131.612,-56.880,-178.895,6.842,148.941
C02768=1144.488,131.881,-56.901,-178.892,6.843,148.941
C02769=1144.483,132.149,-56.924,-178.889,6.846,148.941
C02770=1144.478,132.398,-56.943,-178.886,6.847,148.940
C02771=1144.473,132.647,-56.963,-178.884,6.849,148.940
C02772=1144.468,132.896,-56.983,-178.881,6.851,148.939
C02773=1144.464,133.145,-57.003,-178.878,6.853,148.939
C02774=1144.459,133.395,-57.023,-178.875,6.854,148.939
C02775=1144.455,133.644,-57.043,-178.873,6.856,148.938
C02776=1144.449,133.892,-57.064,-178.870,6.858,148.938
C02777=1144.444,134.142,-57.084,-178.867,6.859,148.937
C02778=1144.440,134.391,-57.104,-178.864,6.862,148.937
C02779=1144.435,134.640,-57.124,-178.861,6.864,148.937
C02780=1144.431,134.889,-57.144,-178.859,6.865,148.936
C02781=1144.426,135.139,-57.165,-178.856,6.867,148.936
C02782=1144.421,135.388,-57.185,-178.853,6.869,148.936
C02783=1144.416,135.637,-57.205,-178.850,6.870,148.935
C02784=1144.411,135.885,-57.225,-178.848,6.872,148.935
C02785=1144.406,136.135,-57.246,-178.845,6.874,148.934
C02786=1144.401,136.384,-57.266,-178.842,6.877,148.934
C02787=1144.397,136.633,-57.286,-178.839,6.878,148.934
C02788=1144.393,136.882,-57.306,-178.837,6.880,148.933
C02789=1144.387,137.132,-57.327,-178.834,6.882,148.933
C02790=1144.383,137.381,-57.347,-178.831,6.884,148.933
C02791=1144.378,137.630,-57.367,-178.829,6.885,148.932
C02792=1144.374,137.879,-57.388,-178.826,6.887,148.932
C02793=1144.369,138.128,-57.409,-178.823,6.890,148.931
C02794=1144.364,138.378,-57.428,-178.820,6.891,148.931
C02795=1144.359,138.627,-57.449,-178.817,6.893,148.931
C02796=1144.354,138.876,-57.470,-178.814,6.895,148.930
C02797=1144.350,139.125,-57.490,-178.812,6.896,148.930
C02798=1144.345,139.374,-57.510,-178.809,6.898,148.930
C02799=1144.340,139.622,-57.531,-178.806,6.901,148.929
C02800=1144.335,139.871,-57.551,-178.803,6.902,148.929
C02801=1144.330,140.121,-57.571,-178.800,6.904,148.928
C02802=1144.325,140.370,-57.592,-178.798,6.906,148.928
C02803=1144.321,140.619,-57.612,-178.795,6.907,148.928
C02804=1144.316,140.868,-57.633,-178.792,6.909,148.927
C02805=1144.311,141.117,-57.654,-178.789,6.912,148.927
C02806=1144.307,141.366,-57.674,-178.787,6.914,148.927
C02807=1144.302,141.615,-57.695,-178.784,6.915,148.926
C02808=1144.297,141.864,-57.715,-178.781,6.917,148.926
C02809=1144.293,142.113,-57.736,-178.778,6.919,148.925
C02810=1144.288,142.363,-57.757,-178.776,6.921,148.925
C02811=1144.284,142.612,-57.777,-178.772,6.923,148.925
C02812=1144.278,142.861,-57.798,-178.770,6.925,148.924
C02813=1144.274,143.110,-57.819,-178.767,6.926,148.924
C02814=1144.269,143.360,-57.840,-178.764,6.928,148.924
C02815=1144.264,143.609,-57.860,-178.762,6.930,148.923
C02816=1144.259,143.858,-57.881,-178.758,6.932,148.923
C02817=1144.255,144.107,-57.901,-178.756,6.934,148.922
C02818=1144.250,144.356,-57.922,-178.753,6.936,148.922
C02819=1144.246,144.604,-57.944,-178.751,6.938,148.922
C02820=1144.240,144.854,-57.965,-178.748,6.940,148.921
C02821=1144.236,145.103,-57.985,-178.745,6.942,148.921
C02822=1144.231,145.352,-58.006,-178.742,6.944,148.921
C02823=1144.226,145.601,-58.026,-178.739,6.946,148.920
C02824=1144.221,145.850,-58.047,-178.736,6.947,148.920
C02825=1144.217,146.100,-58.068,-178.734,6.949,148.920
C02826=1144.212,146.348,-58.090,-178.730,6.951,148.919
C02827=1144.208,146.597,-58.110,-178.728,6.954,148.919
C02828=1144.203,146.847,-58.131,-178.725,6.955,148.919
C02829=1144.198,147.096,-58.151,-178.723,6.957,148.918
C02830=1144.193,147.345,-58.172,-178.720,6.959,148.918
C02831=1144.188,147.593,-58.194,-178.717,6.961,148.918
C02832=1144.184,147.842,-58.214,-178.714,6.963,148.917
C02833=1144.179,148.092,-58.235,-178.711,6.965,148.917
C02834=1144.174,148.342,-58.257,-178.709,6.966,148.916
C02835=1144.170,148.590,-58.278,-178.705,6.969,148.916
C02836=1144.165,148.839,-58.299,-178.703,6.971,148.916
C02837=1144.160,149.088,-58.319,-178.700,6.973,148.915
C02838=1144.156,149.337,-58.341,-178.698,6.974,148.915
C02839=1144.150,149.586,-58.362,-178.694,6.977,148.915
C02840=1144.146,149.836,-58.382,-178.692,6.979,148.914
C02841=1144.142,150.084,-58.404,-178.689,6.980,148.914
C02842=1144.136,150.334,-58.425,-178.686,6.982,148.914
C02843=1144.132,150.583,-58.445,-178.683,6.984,148.913
C02844=1144.127,150.831,-58.467,-178.681,6.987,148.913
C02845=1144.123,151.081,-58.488,-178.678,6.988,148.913
C02846=1144.118,151.330,-58.510,-178.675,6.990,148.912
C02847=1144.113,151.579,-58.531,-178.672,6.993,148.912
C02848=1144.108,151.828,-58.552,-178.669,6.994,148.911
C02849=1144.103,152.077,-58.573,-178.667,6.996,148.911
C02850=1144.099,152.327,-58.595,-178.664,6.998,148.911
C02851=1144.095,152.575,-58.616,-178.661,7.001,148.911
C02852=1144.089,152.824,-58.637,-178.658,7.002,148.910
C02853=1144.084,153.073,-58.658,-178.656,7.004,148.910
C02854=1144.080,153.323,-58.680,-178.653,7.006,148.909
C02855=1144.076,153.571,-58.701,-178.650,7.008,148.909
C02856=1144.071,153.820,-58.722,-178.647,7.010,148.909
C02857=1144.066,154.069,-58.743,-178.645,7.012,148.909
C02858=1144.061,154.319,-58.765,-178.642,7.014,148.908
C02859=1144.056,154.568,-58.786,-178.639,7.016,148.908
C02860=1144.051,154.816,-58.808,-178.636,7.018,148.907
C02861=1144.047,155.065,-58.828,-178.633,7.020,148.907
C02862=1144.043,155.315,-58.850,-178.630,7.022,148.907
C02863=1144.038,155.564,-58.871,-178.628,7.024,148.906
C02864=1144.033,155.812,-58.893,-178.625,7.026,148.906
C02865=1144.028,156.062,-58.915,-178.622,7.028,148.906
C02866=1144.023,156.311,-58.936,-178.619,7.030,148.905
C02867=1144.018,156.560,-58.958,-178.616,7.032,148.905
C02868=1144.014,156.808,-58.979,-178.614,7.034,148.905
C02869=1144.010,157.058,-59.000,-178.611,7.037,148.904
C02870=1144.004,157.327,-59.024,-178.608,7.038,148.904
C02871=1144.000,157.596,-59.047,-178.605,7.041,148.904
C02872=1143.994,157.865,-59.070,-178.602,7.043,148.903
C02873=1143.990,158.134,-59.094,-178.599,7.045,148.903
C02874=1143.985,158.383,-59.115,-178.596,7.047,148.903
C02875=1143.980,158.631,-59.137,-178.593,7.049,148.902
C02876=1143.975,158.881,-59.159,-178.590,7.051,148.902
C02877=1143.971,159.129,-59.180,-178.588,7.053,148.902
C02878=1143.965,159.379,-59.201,-178.585,7.055,148.901
C02879=1143.961,159.628,-59.223,-178.582,7.057,148.901
C02880=1143.956,159.877,-59.245,-178.579,7.059,148.901
C02881=1143.952,160.126,-59.267,-178.577,7.061,148.900
C02882=1143.947,160.375,-59.289,-178.574,7.064,148.900
C02883=1143.942,160.623,-59.310,-178.571,7.066,148.900
C02884=1143.938,160.873,-59.332,-178.568,7.067,148.899
C02885=1143.933,161.122,-59.353,-178.565,7.070,148.899
C02886=1143.929,161.371,-59.375,-178.563,7.072,148.899
C02887=1143.924,161.620,-59.397,-178.560,7.074,148.898
C02888=1143.919,161.869,-59.419,-178.557,7.076,148.898
C02889=1143.915,162.118,-59.441,-178.554,7.078,148.898
C02890=1143.910,162.367,-59.463,-178.552,7.080,148.898
C02891=1143.905,162.616,-59.485,-178.548,7.082,148.897
C02892=1143.900,162.865,-59.507,-178.546,7.084,148.897
C02893=1143.896,163.114,-59.529,-178.543,7.086,148.896
C02894=1143.891,163.363,-59.551,-178.540,7.089,148.896
C02895=1143.886,163.611,-59.572,-178.537,7.090,148.896
C02896=1143.882,163.861,-59.594,-178.535,7.092,148.896
C02897=1143.877,164.109,-59.616,-178.531,7.095,148.895
C02898=1143.872,164.359,-59.638,-178.529,7.096,148.895
C02899=1143.868,164.607,-59.660,-178.527,7.099,148.895
C02900=1143.863,164.857,-59.682,-178.523,7.101,148.894
C02901=1143.858,165.106,-59.704,-178.521,7.103,148.894
C02902=1143.853,165.355,-59.726,-178.517,7.105,148.894
C02903=1143.849,165.604,-59.748,-178.515,7.107,148.893
C02904=1143.844,165.853,-59.770,-178.512,7.109,148.893
C02905=1143.840,166.101,-59.792,-178.509,7.112,148.893
C02906=1143.835,166.351,-59.815,-178.507,7.114,148.893
C02907=1143.830,166.599,-59.837,-178.504,7.115,148.892
C02908=1143.826,166.849,-59.859,-178.501,7.118,148.892
C02909=1143.821,167.097,-59.880,-178.498,7.120,148.891
C02910=1143.816,167.347,-59.902,-178.495,7.123,148.891
C02911=1143.811,167.596,-59.925,-178.493,7.124,148.891
C02912=1143.807,167.844,-59.947,-178.490,7.126,148.891
C02913=1143.803,168.094,-59.969,-178.487,7.129,148.890
C02914=1143.798,168.342,-59.991,-178.484,7.131,148.890
C02915=1143.793,168.592,-60.014,-178.482,7.132,148.890
C02916=1143.788,168.840,-60.036,-178.478,7.135,148.889
C02917=1143.784,169.089,-60.058,-178.476,7.137,148.889
C02918=1143.778,169.338,-60.080,-178.473,7.140,148.889
C02919=1143.774,169.588,-60.103,-178.470,7.141,148.888
C02920=1143.770,169.836,-60.125,-178.467,7.143,148.888
C02921=1143.764,170.085,-60.148,-178.465,7.146,148.888
C02922=1143.760,170.335,-60.170,-178.462,7.148,148.888
C02923=1143.756,170.583,-60.192,-178.459,7.150,148.887
C02924=1143.751,170.832,-60.215,-178.456,7.152,148.887
C02925=1143.746,171.082,-60.237,-178.454,7.154,148.887
C02926=1143.742,171.330,-60.259,-178.450,7.157,148.886
C02927=1143.737,171.579,-60.282,-178.448,7.159,148.886
C02928=1143.732,171.827,-60.304,-178.445,7.161,148.886
C02929=1143.728,172.077,-60.326,-178.442,7.163,148.886
C02930=1143.723,172.326,-60.349,-178.439,7.165,148.885
C02931=1143.718,172.574,-60.371,-178.437,7.167,148.885
C02932=1143.713,172.824,-60.394,-178.434,7.169,148.885
C02933=1143.709,173.073,-60.417,-178.431,7.172,148.884
C02934=1143.705,173.321,-60.438,-178.428,7.174,148.884
C02935=1143.700,173.570,-60.462,-178.425,7.176,148.884
C02936=1143.696,173.820,-60.484,-178.422,7.178,148.883
C02937=1143.690,174.068,-60.507,-178.420,7.180,148.883
C02938=1143.686,174.317,-60.529,-178.417,7.183,148.883
C02939=1143.681,174.566,-60.552,-178.414,7.184,148.883
C02940=1143.676,174.815,-60.574,-178.411,7.187,148.882
C02941=1143.672,175.064,-60.597,-178.409,7.189,148.882
C02942=1143.667,175.313,-60.619,-178.405,7.192,148.882
C02943=1143.662,175.562,-60.642,-178.403,7.194,148.882
C02944=1143.658,175.811,-60.665,-178.400,7.196,148.881
C02945=1143.653,176.060,-60.688,-178.397,7.198,148.881
C02946=1143.649,176.309,-60.710,-178.395,7.200,148.881
C02947=1143.644,176.558,-60.733,-178.392,7.203,148.880
C02948=1143.640,176.807,-60.755,-178.389,7.204,148.880
C02949=1143.635,177.056,-60.779,-178.386,7.207,148.880
C02950=1143.631,177.305,-60.801,-178.384,7.209,148.879
C02951=1143.625,177.553,-60.824,-178.381,7.212,148.879
C02952=1143.621,177.802,-60.847,-178.378,7.214,148.879
C02953=1143.616,178.052,-60.869,-178.375,7.216,148.879
C02954=1143.612,178.301,-60.893,-178.372,7.218,148.879
C02955=1143.607,178.549,-60.915,-178.369,7.221,148.878
C02956=1143.602,178.798,-60.938,-178.367,7.222,148.878
C02957=1143.598,179.047,-60.960,-178.364,7.225,148.878
C02958=1143.593,179.296,-60.984,-178.361,7.227,148.877
C02959=1143.588,179.544,-61.007,-178.358,7.229,148.877
C02960=1143.584,179.793,-61.030,-178.355,7.232,148.877
C02961=1143.580,180.042,-61.053,-178.353,7.233,148.876
C02962=1143.575,180.292,-61.076,-178.350,7.236,148.876
C02963=1143.571,180.541,-61.098,-178.347,7.238,148.876
C02964=1143.566,180.790,-61.122,-178.344,7.241,148.876
C02965=1143.561,181.038,-61.145,-178.342,7.243,148.875
C02966=1143.557,181.287,-61.167,-178.338,7.245,148.875
C02967=1143.552,181.536,-61.191,-178.336,7.247,148.875
C02968=1143.547,181.785,-61.214,-178.333,7.250,148.875
C02969=1143.543,182.034,-61.236,-178.330,7.252,148.874
C02970=1143.538,182.283,-61.260,-178.327,7.255,148.874
C02971=1143.533,182.531,-61.283,-178.325,7.256,148.874
C02972=1143.529,182.780,-61.305,-178.322,7.259,148.874
C02973=1143.524,183.029,-61.329,-178.319,7.261,148.873
C02974=1143.519,183.299,-61.354,-178.316,7.263,148.873
C02975=1143.514,183.568,-61.379,-178.313,7.266,148.873
C02976=1143.510,183.838,-61.404,-178.310,7.269,148.873
C02977=1143.505,184.108,-61.429,-178.307,7.271,148.872
C02978=1143.500,184.357,-61.453,-178.304,7.273,148.872
C02979=1143.495,184.605,-61.476,-178.302,7.275,148.872
C02980=1143.490,184.854,-61.499,-178.298,7.278,148.871
C02981=1143.486,185.103,-61.522,-178.296,7.281,148.871
C02982=1143.481,185.352,-61.545,-178.293,7.282,148.871
C02983=1143.477,185.601,-61.568,-178.290,7.285,148.871
C02984=1143.472,185.850,-61.592,-178.287,7.287,148.870
C02985=1143.467,186.099,-61.616,-178.284,7.290,148.870
C02986=1143.463,186.348,-61.639,-178.282,7.292,148.870
C02987=1143.459,186.596,-61.662,-178.279,7.294,148.870
C02988=1143.454,186.845,-61.685,-178.276,7.296,148.869
C02989=1143.449,187.094,-61.709,-178.273,7.299,148.869
C02990=1143.445,187.343,-61.732,-178.271,7.301,148.869
C02991=1143.440,187.593,-61.755,-178.268,7.304,148.869
C02992=1143.436,187.841,-61.780,-178.265,7.306,148.868
C02993=1143.431,188.090,-61.803,-178.262,7.308,148.868
C02994=1143.426,188.338,-61.826,-178.260,7.310,148.868
C02995=1143.421,188.587,-61.849,-178.257,7.313,148.868
C02996=1143.416,188.836,-61.873,-178.253,7.315,148.867
C02997=1143.412,189.085,-61.897,-178.251,7.317,148.867
C02998=1143.407,189.334,-61.920,-178.248,7.320,148.867
C02999=1143.402,189.583,-61.943,-178.246,7.322,148.867
C03000=1143.398,189.831,-61.967,-178.242,7.325,148.866
C03001=1143.393,190.080,-61.991,-178.240,7.327,148.866
C03002=1143.389,190.329,-62.014,-178.237,7.329,148.866
C03003=1143.384,190.578,-62.038,-178.235,7.331,148.866
C03004=1143.380,190.827,-62.062,-178.231,7.334,148.865
C03005=1143.375,191.076,-62.085,-178.228,7.337,148.865
C03006=1143.370,191.324,-62.109,-178.226,7.339,148.865
C03007=1143.366,191.574,-62.133,-178.223,7.341,148.865
C03008=1143.362,191.823,-62.156,-178.220,7.343,148.864
C03009=1143.357,192.071,-62.180,-178.217,7.346,148.864
C03010=1143.353,192.320,-62.204,-178.215,7.348,148.864
C03011=1143.348,192.569,-62.228,-178.212,7.351,148.864
C03012=1143.343,192.818,-62.251,-178.209,7.353,148.864
C03013=1143.339,193.067,-62.274,-178.206,7.355,148.863
C03014=1143.334,193.315,-62.298,-178.203,7.358,148.863
C03015=1143.330,193.564,-62.322,-178.201,7.360,148.863
C03016=1143.325,193.813,-62.346,-178.198,7.363,148.863
C03017=1143.321,194.062,-62.369,-178.195,7.365,148.862
C03018=1143.316,194.310,-62.393,-178.192,7.367,148.862
C03019=1143.311,194.560,-62.417,-178.189,7.370,148.862
C03020=1143.307,194.809,-62.442,-178.187,7.372,148.862
C03021=1143.303,195.057,-62.466,-178.184,7.375,148.862
C03022=1143.298,195.306,-62.489,-178.181,7.376,148.861
C03023=1143.293,195.554,-62.513,-178.178,7.379,148.861
C03024=1143.289,195.804,-62.537,-178.175,7.382,148.861
C03025=1143.284,196.052,-62.561,-178.173,7.384,148.861
C03026=1143.279,196.301,-62.585,-178.170,7.387,148.860
C03027=1143.275,196.550,-62.609,-178.167,7.389,148.860
C03028=1143.271,196.799,-62.633,-178.164,7.391,148.860
C03029=1143.266,197.048,-62.656,-178.161,7.394,148.860
C03030=1143.261,197.297,-62.681,-178.159,7.396,148.859
C03031=1143.257,197.545,-62.705,-178.156,7.399,148.859
C03032=1143.252,197.794,-62.729,-178.153,7.402,148.859
C03033=1143.247,198.042,-62.753,-178.150,7.403,148.859
C03034=1143.243,198.292,-62.778,-178.148,7.406,148.859
C03035=1143.239,198.540,-62.802,-178.145,7.408,148.858
C03036=1143.234,198.789,-62.825,-178.142,7.411,148.858
C03037=1143.229,199.038,-62.849,-178.139,7.413,148.858
C03038=1143.224,199.286,-62.874,-178.137,7.416,148.858
C03039=1143.220,199.536,-62.898,-178.133,7.418,148.857
C03040=1143.216,199.785,-62.922,-178.130,7.421,148.857
C03041=1143.211,200.033,-62.946,-178.128,7.423,148.857
C03042=1143.206,200.282,-62.970,-178.125,7.426,148.857
C03043=1143.202,200.531,-62.995,-178.122,7.429,148.857
C03044=1143.197,200.780,-63.019,-178.119,7.430,148.856
C03045=1143.193,201.028,-63.044,-178.117,7.433,148.856
C03046=1143.188,201.277,-63.067,-178.114,7.435,148.856
C03047=1143.184,201.526,-63.092,-178.111,7.438,148.856
C03048=1143.179,201.775,-63.116,-178.108,7.441,148.856
C03049=1143.175,202.023,-63.140,-178.106,7.443,148.855
C03050=1143.170,202.272,-63.165,-178.103,7.445,148.855
C03051=1143.166,202.521,-63.189,-178.100,7.448,148.855
C03052=1143.162,202.769,-63.213,-178.097,7.450,148.855
C03053=1143.156,203.018,-63.238,-178.095,7.453,148.855
C03054=1143.153,203.267,-63.262,-178.091,7.456,148.854
C03055=1143.148,203.516,-63.287,-178.089,7.458,148.854
C03056=1143.143,203.764,-63.311,-178.086,7.460,148.854
C03057=1143.138,204.013,-63.336,-178.083,7.463,148.854
C03058=1143.134,204.262,-63.360,-178.081,7.465,148.854
C03059=1143.129,204.511,-63.385,-178.077,7.468,148.853
C03060=1143.125,204.759,-63.409,-178.075,7.471,148.853
C03061=1143.120,205.009,-63.434,-178.072,7.472,148.853
C03062=1143.116,205.257,-63.458,-178.069,7.475,148.853
C03063=1143.111,205.506,-63.483,-178.066,7.478,148.853
C03064=1143.107,205.755,-63.507,-178.064,7.480,148.852
C03065=1143.102,206.004,-63.532,-178.061,7.483,148.852
C03066=1143.098,206.252,-63.557,-178.058,7.486,148.852
C03067=1143.093,206.501,-63.582,-178.055,7.488,148.852
C03068=1143.089,206.749,-63.606,-178.053,7.490,148.852
C03069=1143.084,206.998,-63.630,-178.050,7.493,148.852
C03070=1143.080,207.247,-63.655,-178.047,7.496,148.851
C03071=1143.075,207.496,-63.680,-178.044,7.498,148.851
C03072=1143.071,207.745,-63.705,-178.041,7.501,148.851
C03073=1143.066,207.993,-63.729,-178.038,7.503,148.851
C03074=1143.061,208.242,-63.754,-178.036,7.506,148.851
C03075=1143.057,208.491,-63.779,-178.033,7.508,148.850
C03076=1143.052,208.739,-63.804,-178.030,7.511,148.850
C03077=1143.048,208.988,-63.828,-178.028,7.513,148.850
C03078=1143.043,209.259,-63.856,-178.024,7.516,148.850
C03079=1143.038,209.530,-63.883,-178.021,7.519,148.850
C03080=1143.033,209.800,-63.909,-178.018,7.522,148.849
C03081=1143.028,210.071,-63.937,-178.015,7.525,148.849
C03082=1143.023,210.319,-63.961,-178.013,7.527,148.849
C03083=1143.020,210.568,-63.986,-178.010,7.530,148.849
C03084=1143.015,210.817,-64.011,-178.007,7.532,148.849
C03085=1143.010,211.066,-64.036,-178.004,7.535,148.849
C03086=1143.006,211.314,-64.061,-178.001,7.537,148.848
C03087=1143.001,211.563,-64.086,-177.998,7.540,148.848
C03088=1142.996,211.812,-64.111,-177.996,7.543,148.848
C03089=1142.992,212.061,-64.136,-177.993,7.545,148.848
C03090=1142.988,212.309,-64.160,-177.990,7.548,148.848
C03091=1142.983,212.557,-64.186,-177.987,7.550,148.847
C03092=1142.978,212.807,-64.211,-177.984,7.553,148.847
C03093=1142.974,213.055,-64.236,-177.982,7.555,148.847
C03094=1142.970,213.304,-64.261,-177.979,7.558,148.847
C03095=1142.965,213.553,-64.286,-177.976,7.561,148.847
C03096=1142.960,213.801,-64.311,-177.973,7.564,148.847
C03097=1142.956,214.050,-64.337,-177.971,7.566,148.846
C03098=1142.951,214.299,-64.361,-177.968,7.569,148.846
C03099=1142.948,214.548,-64.387,-177.965,7.571,148.846
C03100=1142.942,214.796,-64.411,-177.962,7.574,148.846
C03101=1142.938,215.045,-64.437,-177.960,7.576,148.846
C03102=1142.933,215.293,-64.462,-177.957,7.579,148.846
C03103=1142.929,215.543,-64.487,-177.954,7.582,148.845
C03104=1142.925,215.790,-64.512,-177.951,7.584,148.845
C03105=1142.920,216.039,-64.538,-177.949,7.587,148.845
C03106=1142.916,216.289,-64.563,-177.945,7.589,148.845
C03107=1142.911,216.537,-64.588,-177.943,7.592,148.845
C03108=1142.907,216.786,-64.614,-177.940,7.595,148.845
C03109=1142.902,217.034,-64.639,-177.937,7.597,148.845
C03110=1142.898,217.283,-64.665,-177.934,7.600,148.844
C03111=1142.893,217.531,-64.690,-177.931,7.603,148.844
C03112=1142.888,217.781,-64.715,-177.929,7.605,148.844
C03113=1142.885,218.029,-64.740,-177.926,7.608,148.844
C03114=1142.880,218.277,-64.766,-177.923,7.610,148.844
C03115=1142.876,218.526,-64.791,-177.920,7.613,148.843
C03116=1142.871,218.775,-64.816,-177.918,7.616,148.843
C03117=1142.866,219.023,-64.842,-177.915,7.619,148.843
C03118=1142.862,219.272,-64.867,-177.913,7.621,148.843
C03119=1142.857,219.520,-64.893,-177.909,7.623,148.843
C03120=1142.853,219.769,-64.919,-177.906,7.626,148.843
C03121=1142.848,220.019,-64.944,-177.904,7.629,148.843
C03122=1142.844,220.267,-64.969,-177.901,7.632,148.843
C03123=1142.839,220.516,-64.995,-177.898,7.634,148.842
C03124=1142.835,220.764,-65.021,-177.895,7.637,148.842
C03125=1142.830,221.012,-65.046,-177.893,7.640,148.842
C03126=1142.826,221.261,-65.072,-177.890,7.643,148.842
C03127=1142.822,221.510,-65.097,-177.887,7.645,148.842
C03128=1142.817,221.758,-65.123,-177.884,7.647,148.842
C03129=1142.813,222.007,-65.149,-177.881,7.650,148.841
C03130=1142.808,222.256,-65.175,-177.879,7.653,148.841
C03131=1142.804,222.505,-65.201,-177.876,7.656,148.841
C03132=1142.799,222.753,-65.226,-177.873,7.659,148.841
C03133=1142.795,223.002,-65.252,-177.870,7.662,148.841
C03134=1142.790,223.251,-65.278,-177.868,7.664,148.841
C03135=1142.786,223.499,-65.303,-177.865,7.667,148.841
C03136=1142.781,223.747,-65.329,-177.862,7.670,148.841
C03137=1142.777,223.996,-65.354,-177.859,7.672,148.840
C03138=1142.773,224.245,-65.380,-177.856,7.675,148.840
C03139=1142.767,224.494,-65.406,-177.853,7.678,148.840
C03140=1142.763,224.742,-65.432,-177.851,7.680,148.840
C03141=1142.759,224.991,-65.458,-177.848,7.683,148.840
C03142=1142.755,225.240,-65.483,-177.845,7.686,148.840
C03143=1142.750,225.488,-65.509,-177.842,7.688,148.839
C03144=1142.745,225.737,-65.536,-177.839,7.691,148.839
C03145=1142.741,225.985,-65.562,-177.836,7.694,148.839
C03146=1142.737,226.234,-65.587,-177.834,7.696,148.839
C03147=1142.733,226.483,-65.613,-177.831,7.699,148.839
C03148=1142.728,226.731,-65.638,-177.829,7.702,148.839
C03149=1142.723,226.980,-65.665,-177.825,7.705,148.839
C03150=1142.719,227.228,-65.691,-177.823,7.708,148.839
C03151=1142.715,227.477,-65.717,-177.820,7.711,148.838
C03152=1142.710,227.726,-65.743,-177.818,7.713,148.838
C03153=1142.705,227.974,-65.769,-177.815,7.716,148.838
C03154=1142.701,228.223,-65.795,-177.812,7.718,148.838
C03155=1142.697,228.471,-65.821,-177.809,7.721,148.838
C03156=1142.692,228.720,-65.847,-177.806,7.724,148.838
C03157=1142.688,228.969,-65.874,-177.803,7.727,148.838
C03158=1142.684,229.217,-65.900,-177.800,7.730,148.838
C03159=1142.679,229.467,-65.926,-177.798,7.732,148.838
C03160=1142.674,229.714,-65.952,-177.795,7.735,148.837
C03161=1142.670,229.963,-65.978,-177.793,7.738,148.837
C03162=1142.665,230.212,-66.004,-177.790,7.741,148.837
C03163=1142.661,230.460,-66.031,-177.786,7.743,148.837
C03164=1142.657,230.709,-66.056,-177.784,7.746,148.837
C03165=1142.652,230.957,-66.083,-177.781,7.749,148.837
C03166=1142.648,231.206,-66.109,-177.778,7.752,148.837
C03167=1142.644,231.454,-66.136,-177.776,7.754,148.837
C03168=1142.638,231.703,-66.162,-177.773,7.757,148.836
C03169=1142.634,231.951,-66.188,-177.770,7.760,148.836
C03170=1142.630,232.200,-66.214,-177.767,7.763,148.836
C03171=1142.626,232.448,-66.241,-177.764,7.765,148.836
C03172=1142.621,232.697,-66.267,-177.761,7.768,148.836
C03173=1142.617,232.946,-66.294,-177.759,7.771,148.836
C03174=1142.612,233.194,-66.319,-177.756,7.774,148.836
C03175=1142.608,233.443,-66.346,-177.753,7.777,148.836
C03176=1142.604,233.692,-66.372,-177.751,7.779,148.836
C03177=1142.599,233.940,-66.399,-177.748,7.782,148.835
C03178=1142.595,234.189,-66.425,-177.745,7.785,148.835
C03179=1142.590,234.438,-66.452,-177.742,7.788,148.835
C03180=1142.586,234.686,-66.479,-177.740,7.791,148.835
C03181=1142.581,234.935,-66.505,-177.737,7.794,148.835
C03182=1142.576,235.206,-66.534,-177.734,7.796,148.835
C03183=1142.572,235.478,-66.563,-177.730,7.800,148.835
C03184=1142.567,235.751,-66.592,-177.727,7.803,148.835
C03185=1142.562,236.022,-66.621,-177.725,7.806,148.835
C03186=1142.558,236.270,-66.648,-177.722,7.809,148.835
C03187=1142.553,236.520,-66.674,-177.719,7.812,148.834
C03188=1142.549,236.768,-66.701,-177.716,7.815,148.834
C03189=1142.544,237.016,-66.728,-177.713,7.818,148.834
C03190=1142.540,237.265,-66.755,-177.710,7.820,148.834
C03191=1142.536,237.513,-66.781,-177.707,7.823,148.834
C03192=1142.531,237.762,-66.808,-177.705,7.826,148.834
C03193=1142.527,238.010,-66.834,-177.702,7.828,148.834
C03194=1142.522,238.259,-66.861,-177.700,7.831,148.834
C03195=1142.517,238.507,-66.888,-177.697,7.834,148.834
C03196=1142.514,238.755,-66.915,-177.694,7.837,148.833
C03197=1142.509,239.005,-66.941,-177.691,7.840,148.833
C03198=1142.504,239.253,-66.968,-177.688,7.843,148.833
C03199=1142.500,239.501,-66.995,-177.686,7.846,148.833
C03200=1142.495,239.750,-67.022,-177.683,7.848,148.833
C03201=1142.491,239.999,-67.049,-177.680,7.851,148.833
C03202=1142.487,240.247,-67.076,-177.677,7.854,148.833
C03203=1142.483,240.496,-67.103,-177.674,7.857,148.833
C03204=1142.478,240.744,-67.130,-177.672,7.860,148.833
C03205=1142.473,240.993,-67.157,-177.669,7.863,148.833
C03206=1142.470,241.241,-67.183,-177.666,7.866,148.833
C03207=1142.465,241.489,-67.210,-177.663,7.869,148.833
C03208=1142.460,241.738,-67.237,-177.660,7.872,148.833
C03209=1142.456,241.986,-67.264,-177.658,7.875,148.832
C03210=1142.451,242.235,-67.292,-177.655,7.878,148.832
C03211=1142.448,242.484,-67.318,-177.653,7.880,148.832
C03212=1142.443,242.732,-67.345,-177.650,7.883,148.832
C03213=1142.438,242.981,-67.372,-177.647,7.886,148.832
C03214=1142.434,243.229,-67.399,-177.644,7.889,148.832
C03215=1142.429,243.478,-67.426,-177.641,7.891,148.832
C03216=1142.425,243.726,-67.453,-177.639,7.894,148.832
C03217=1142.421,243.975,-67.480,-177.636,7.897,148.832
C03218=1142.417,244.223,-67.508,-177.633,7.900,148.832
C03219=1142.412,244.471,-67.535,-177.630,7.903,148.832
C03220=1142.407,244.720,-67.562,-177.627,7.906,148.832
C03221=1142.403,244.968,-67.589,-177.625,7.909,148.832
C03222=1142.399,245.217,-67.616,-177.622,7.912,148.831
C03223=1142.395,245.465,-67.644,-177.619,7.915,148.831
C03224=1142.390,245.714,-67.671,-177.616,7.918,148.831
C03225=1142.386,245.962,-67.698,-177.614,7.921,148.831
C03226=1142.381,246.211,-67.725,-177.611,7.924,148.831
C03227=1142.377,246.459,-67.753,-177.608,7.926,148.831
C03228=1142.373,246.708,-67.780,-177.605,7.929,148.831
C03229=1142.368,246.956,-67.807,-177.602,7.932,148.831
C03230=1142.363,247.205,-67.834,-177.600,7.935,148.831
C03231=1142.360,247.453,-67.863,-177.597,7.938,148.831
C03232=1142.355,247.702,-67.890,-177.594,7.941,148.831
C03233=1142.350,247.950,-67.917,-177.591,7.944,148.831
C03234=1142.346,248.198,-67.944,-177.588,7.947,148.831
C03235=1142.342,248.447,-67.972,-177.586,7.950,148.830
C03236=1142.337,248.696,-67.999,-177.583,7.953,148.830
C03237=1142.333,248.944,-68.027,-177.580,7.956,148.830
C03238=1142.329,249.193,-68.054,-177.577,7.959,148.830
C03239=1142.324,249.441,-68.082,-177.574,7.961,148.830
C03240=1142.320,249.689,-68.109,-177.572,7.964,148.830
C03241=1142.315,249.937,-68.137,-177.569,7.967,148.830
C03242=1142.311,250.186,-68.164,-177.566,7.971,148.830
C03243=1142.307,250.434,-68.192,-177.564,7.974,148.830
C03244=1142.302,250.683,-68.219,-177.561,7.976,148.830
C03245=1142.299,250.931,-68.247,-177.558,7.979,148.830
C03246=1142.294,251.180,-68.274,-177.555,7.982,148.830
C03247=1142.290,251.428,-68.302,-177.553,7.985,148.830
C03248=1142.285,251.677,-68.330,-177.550,7.988,148.830
C03249=1142.280,251.925,-68.358,-177.547,7.991,148.830
C03250=1142.276,252.174,-68.385,-177.544,7.994,148.830
C03251=1142.272,252.422,-68.413,-177.541,7.997,148.830
C03252=1142.268,252.670,-68.441,-177.539,8.000,148.829
C03253=1142.264,252.919,-68.468,-177.536,8.003,148.829
C03254=1142.259,253.167,-68.496,-177.533,8.006,148.829
C03255=1142.254,253.416,-68.524,-177.531,8.009,148.829
C03256=1142.250,253.664,-68.552,-177.528,8.012,148.829
C03257=1142.246,253.912,-68.580,-177.525,8.015,148.829
C03258=1142.241,254.161,-68.607,-177.522,8.018,148.829
C03259=1142.237,254.409,-68.635,-177.519,8.021,148.829
C03260=1142.232,254.658,-68.663,-177.517,8.024,148.829
C03261=1142.229,254.906,-68.691,-177.514,8.026,148.829
C03262=1142.224,255.155,-68.718,-177.511,8.030,148.829
C03263=1142.220,255.403,-68.746,-177.508,8.033,148.829
C03264=1142.215,255.651,-68.775,-177.505,8.036,148.829
C03265=1142.211,255.899,-68.803,-177.503,8.039,148.829
C03266=1142.207,256.148,-68.830,-177.500,8.042,148.829
C03267=1142.202,256.396,-68.858,-177.497,8.045,148.829
C03268=1142.198,256.645,-68.887,-177.494,8.048,148.829
C03269=1142.193,256.893,-68.914,-177.491,8.051,148.829
C03270=1142.190,257.142,-68.943,-177.489,8.054,148.829
C03271=1142.185,257.390,-68.971,-177.486,8.057,148.829
C03272=1142.181,257.638,-68.999,-177.484,8.060,148.829
C03273=1142.176,257.887,-69.026,-177.481,8.063,148.829
C03274=1142.172,258.136,-69.055,-177.478,8.066,148.829
C03275=1142.167,258.384,-69.083,-177.475,8.069,148.829
C03276=1142.164,258.632,-69.111,-177.472,8.072,148.829
C03277=1142.159,258.880,-69.139,-177.470,8.075,148.828
C03278=1142.155,259.129,-69.167,-177.467,8.078,148.828
C03279=1142.150,259.377,-69.195,-177.464,8.082,148.829
C03280=1142.146,259.626,-69.224,-177.461,8.085,148.829
C03281=1142.142,259.874,-69.252,-177.458,8.088,148.828
C03282=1142.137,260.123,-69.280,-177.456,8.090,148.828
C03283=1142.133,260.370,-69.308,-177.453,8.093,148.828
C03284=1142.129,260.619,-69.336,-177.450,8.096,148.828
C03285=1142.124,260.867,-69.365,-177.448,8.100,148.828
C03286=1142.120,261.141,-69.396,-177.445,8.102,148.828
C03287=1142.115,261.414,-69.428,-177.441,8.106,148.828
C03288=1142.110,261.688,-69.458,-177.439,8.109,148.828
C03289=1142.105,261.961,-69.490,-177.435,8.113,148.828
C03290=1142.101,262.210,-69.518,-177.432,8.116,148.828
C03291=1142.096,262.458,-69.546,-177.430,8.119,148.828
C03292=1142.092,262.706,-69.575,-177.427,8.122,148.828
C03293=1142.088,262.955,-69.604,-177.425,8.125,148.828
C03294=1142.084,263.203,-69.631,-177.422,8.128,148.828
C03295=1142.079,263.452,-69.660,-177.418,8.132,148.828
C03296=1142.075,263.699,-69.688,-177.416,8.135,148.828
C03297=1142.071,263.948,-69.717,-177.413,8.138,148.828
C03298=1142.067,264.196,-69.746,-177.410,8.141,148.828
C03299=1142.062,264.445,-69.774,-177.408,8.144,148.828
C03300=1142.057,264.693,-69.803,-177.405,8.147,148.828
C03301=1142.054,264.941,-69.832,-177.403,8.150,148.828
C03302=1142.049,265.190,-69.860,-177.400,8.153,148.828
C03303=1142.045,265.438,-69.888,-177.397,8.156,148.828
C03304=1142.040,265.686,-69.917,-177.394,8.159,148.828
C03305=1142.036,265.935,-69.946,-177.391,8.162,148.828
C03306=1142.032,266.183,-69.974,-177.388,8.166,148.828
C03307=1142.027,266.431,-70.003,-177.386,8.169,148.828
C03308=1142.023,266.680,-70.032,-177.383,8.171,148.828
C03309=1142.019,266.928,-70.060,-177.380,8.174,148.828
C03310=1142.014,267.176,-70.089,-177.378,8.178,148.828
C03311=1142.010,267.425,-70.118,-177.375,8.181,148.828
C03312=1142.006,267.673,-70.147,-177.372,8.183,148.828
C03313=1142.002,267.921,-70.175,-177.369,8.187,148.828
C03314=1141.997,268.169,-70.204,-177.367,8.190,148.828
C03315=1141.993,268.418,-70.233,-177.364,8.193,148.828
C03316=1141.989,268.666,-70.262,-177.361,8.196,148.828
C03317=1141.984,268.914,-70.290,-177.358,8.199,148.828
C03318=1141.980,269.162,-70.320,-177.356,8.203,148.828
C03319=1141.976,269.411,-70.348,-177.353,8.205,148.828
C03320=1141.972,269.659,-70.378,-177.350,8.208,148.828
C03321=1141.967,269.907,-70.406,-177.347,8.212,148.828
C03322=1141.962,270.156,-70.435,-177.345,8.215,148.828
C03323=1141.959,270.404,-70.463,-177.342,8.218,148.828
C03324=1141.955,270.652,-70.493,-177.339,8.221,148.828
C03325=1141.950,270.900,-70.522,-177.337,8.224,148.828
C03326=1141.945,271.149,-70.551,-177.334,8.227,148.828
C03327=1141.941,271.397,-70.580,-177.331,8.230,148.828
C03328=1141.938,271.645,-70.609,-177.328,8.234,148.828
C03329=1141.933,271.894,-70.638,-177.325,8.237,148.828
C03330=1141.928,272.142,-70.667,-177.323,8.240,148.828
C03331=1141.924,272.390,-70.696,-177.320,8.243,148.828
C03332=1141.920,272.639,-70.725,-177.317,8.246,148.828
C03333=1141.916,272.887,-70.755,-177.315,8.249,148.828
C03334=1141.911,273.135,-70.784,-177.311,8.253,148.828
C03335=1141.907,273.383,-70.813,-177.309,8.256,148.828
C03336=1141.903,273.631,-70.841,-177.306,8.259,148.828
C03337=1141.899,273.880,-70.871,-177.303,8.262,148.828
C03338=1141.894,274.128,-70.900,-177.301,8.265,148.828
C03339=1141.890,274.376,-70.930,-177.298,8.268,148.828
C03340=1141.886,274.625,-70.959,-177.295,8.272,148.828
C03341=1141.881,274.873,-70.987,-177.293,8.275,148.828
C03342=1141.877,275.121,-71.017,-177.290,8.278,148.828
C03343=1141.873,275.369,-71.046,-177.287,8.281,148.828
C03344=1141.868,275.618,-71.076,-177.285,8.285,148.828
C03345=1141.864,275.866,-71.105,-177.282,8.287,148.828
C03346=1141.860,276.114,-71.135,-177.278,8.291,148.828
C03347=1141.856,276.362,-71.164,-177.276,8.294,148.829
C03348=1141.852,276.611,-71.194,-177.273,8.297,148.829
C03349=1141.848,276.859,-71.223,-177.271,8.300,148.828
C03350=1141.843,277.106,-71.252,-177.268,8.304,148.829
C03351=1141.839,277.355,-71.282,-177.265,8.307,148.829
C03352=1141.834,277.603,-71.311,-177.263,8.311,148.829
C03353=1141.830,277.851,-71.340,-177.260,8.314,148.829
C03354=1141.826,278.099,-71.370,-177.257,8.316,148.829
C03355=1141.822,278.348,-71.399,-177.255,8.320,148.829
C03356=1141.818,278.596,-71.429,-177.252,8.323,148.829
C03357=1141.814,278.844,-71.458,-177.248,8.326,148.829
C03358=1141.809,279.093,-71.488,-177.246,8.330,148.829
C03359=1141.805,279.341,-71.517,-177.243,8.333,148.829
C03360=1141.800,279.589,-71.547,-177.241,8.336,148.829
C03361=1141.796,279.838,-71.577,-177.238,8.339,148.829
C03362=1141.792,280.086,-71.606,-177.235,8.342,148.829
C03363=1141.788,280.334,-71.636,-177.232,8.346,148.829
C03364=1141.784,280.582,-71.666,-177.230,8.349,148.829
C03365=1141.780,280.830,-71.695,-177.227,8.352,148.829
C03366=1141.775,281.078,-71.725,-177.224,8.356,148.829
C03367=1141.771,281.327,-71.755,-177.221,8.359,148.829
C03368=1141.766,281.575,-71.784,-177.219,8.362,148.829
C03369=1141.762,281.823,-71.814,-177.216,8.365,148.829
C03370=1141.758,282.071,-71.844,-177.214,8.368,148.829
C03371=1141.753,282.320,-71.874,-177.210,8.372,148.829
C03372=1141.749,282.567,-71.904,-177.208,8.375,148.830
C03373=1141.745,282.816,-71.933,-177.205,8.378,148.830
C03374=1141.741,283.064,-71.963,-177.202,8.381,148.830
C03375=1141.737,283.312,-71.992,-177.200,8.384,148.830
C03376=1141.732,283.560,-72.023,-177.197,8.388,148.830
C03377=1141.728,283.808,-72.053,-177.194,8.391,148.830
C03378=1141.724,284.057,-72.082,-177.192,8.394,148.830
C03379=1141.719,284.305,-72.113,-177.189,8.397,148.830
C03380=1141.715,284.553,-72.142,-177.186,8.401,148.830
C03381=1141.711,284.801,-72.172,-177.184,8.404,148.830
C03382=1141.706,285.049,-72.202,-177.181,8.407,148.830
C03383=1141.702,285.297,-72.232,-177.179,8.411,148.830
C03384=1141.699,285.546,-72.262,-177.175,8.414,148.830
C03385=1141.694,285.794,-72.293,-177.173,8.418,148.830
C03386=1141.690,286.042,-72.323,-177.170,8.421,148.830
C03387=1141.686,286.290,-72.352,-177.168,8.424,148.831
C03388=1141.681,286.538,-72.383,-177.164,8.428,148.830
C03389=1141.677,286.786,-72.412,-177.162,8.431,148.831
C03390=1141.673,287.062,-72.446,-177.159,8.435,148.831
C03391=1141.668,287.337,-72.480,-177.156,8.437,148.831
C03392=1141.663,287.613,-72.513,-177.153,8.442,148.831
C03393=1141.659,287.888,-72.546,-177.150,8.445,148.831
C03394=1141.654,288.136,-72.576,-177.147,8.449,148.831
C03395=1141.651,288.385,-72.607,-177.144,8.451,148.831
C03396=1141.646,288.633,-72.638,-177.141,8.456,148.831
C03397=1141.642,288.881,-72.667,-177.139,8.458,148.831
C03398=1141.637,289.129,-72.698,-177.136,8.462,148.831
C03399=1141.633,289.377,-72.728,-177.134,8.465,148.831
C03400=1141.628,289.625,-72.758,-177.131,8.469,148.831
C03401=1141.625,289.874,-72.789,-177.128,8.472,148.831
C03402=1141.620,290.122,-72.819,-177.126,8.475,148.832
C03403=1141.617,290.369,-72.850,-177.123,8.478,148.832
C03404=1141.612,290.618,-72.880,-177.120,8.482,148.832
C03405=1141.608,290.865,-72.910,-177.118,8.485,148.832
C03406=1141.604,291.114,-72.941,-177.115,8.488,148.832
C03407=1141.600,291.362,-72.971,-177.112,8.491,148.832
C03408=1141.595,291.610,-73.001,-177.109,8.495,148.832
C03409=1141.591,291.858,-73.031,-177.107,8.498,148.832
C03410=1141.587,292.107,-73.062,-177.104,8.501,148.832
C03411=1141.583,292.354,-73.093,-177.101,8.505,148.832
C03412=1141.579,292.602,-73.123,-177.099,8.509,148.833
C03413=1141.574,292.850,-73.154,-177.096,8.512,148.832
C03414=1141.570,293.099,-73.184,-177.094,8.515,148.833
C03415=1141.566,293.347,-73.215,-177.090,8.519,148.833
C03416=1141.562,293.595,-73.245,-177.088,8.522,148.833
C03417=1141.557,293.843,-73.276,-177.085,8.525,148.833
C03418=1141.553,294.091,-73.307,-177.082,8.529,148.833
C03419=1141.549,294.339,-73.337,-177.080,8.532,148.833
C03420=1141.545,294.587,-73.368,-177.077,8.535,148.833
C03421=1141.541,294.836,-73.399,-177.074,8.539,148.833
C03422=1141.537,295.083,-73.429,-177.071,8.542,148.833
C03423=1141.532,295.331,-73.460,-177.069,8.545,148.833
C03424=1141.528,295.580,-73.491,-177.067,8.549,148.834
C03425=1141.524,295.828,-73.521,-177.063,8.552,148.834
C03426=1141.520,296.075,-73.552,-177.061,8.556,148.834
C03427=1141.516,296.324,-73.583,-177.059,8.559,148.834
C03428=1141.511,296.572,-73.614,-177.055,8.563,148.834
C03429=1141.507,296.820,-73.644,-177.053,8.566,148.834
C03430=1141.504,297.068,-73.676,-177.050,8.569,148.834
C03431=1141.499,297.316,-73.706,-177.047,8.573,148.834
C03432=1141.494,297.564,-73.737,-177.045,8.576,148.834
C03433=1141.491,297.812,-73.768,-177.042,8.579,148.834
C03434=1141.486,298.060,-73.798,-177.039,8.583,148.835
C03435=1141.482,298.309,-73.830,-177.037,8.586,148.835
C03436=1141.478,298.557,-73.860,-177.034,8.589,148.835
C03437=1141.474,298.804,-73.892,-177.031,8.593,148.835
C03438=1141.470,299.052,-73.922,-177.029,8.597,148.835
C03439=1141.466,299.300,-73.953,-177.026,8.600,148.835
C03440=1141.461,299.548,-73.984,-177.023,8.604,148.835
C03441=1141.457,299.796,-74.016,-177.021,8.607,148.836
C03442=1141.453,300.044,-74.047,-177.018,8.610,148.836
C03443=1141.449,300.293,-74.078,-177.015,8.614,148.836
C03444=1141.444,300.540,-74.109,-177.013,8.617,148.836
C03445=1141.441,300.789,-74.140,-177.010,8.620,148.836
C03446=1141.437,301.037,-74.170,-177.007,8.624,148.836
C03447=1141.432,301.284,-74.202,-177.005,8.627,148.836
C03448=1141.428,301.533,-74.233,-177.002,8.631,148.836
C03449=1141.424,301.780,-74.264,-176.999,8.634,148.836
C03450=1141.420,302.029,-74.296,-176.997,8.638,148.837
C03451=1141.415,302.276,-74.326,-176.994,8.641,148.837
C03452=1141.412,302.524,-74.358,-176.991,8.645,148.837
C03453=1141.407,302.772,-74.389,-176.989,8.648,148.837
C03454=1141.403,303.021,-74.420,-176.986,8.652,148.837
C03455=1141.399,303.268,-74.452,-176.983,8.655,148.837
C03456=1141.395,303.517,-74.483,-176.981,8.658,148.837
C03457=1141.390,303.764,-74.514,-176.978,8.662,148.838
C03458=1141.386,304.013,-74.545,-176.975,8.666,148.838
C03459=1141.382,304.260,-74.577,-176.973,8.669,148.838
C03460=1141.378,304.509,-74.608,-176.970,8.673,148.838
C03461=1141.374,304.756,-74.639,-176.967,8.676,148.838
C03462=1141.370,305.004,-74.671,-176.965,8.679,148.838
C03463=1141.365,305.252,-74.702,-176.962,8.683,148.838
C03464=1141.362,305.500,-74.734,-176.959,8.686,148.838
C03465=1141.357,305.748,-74.765,-176.956,8.690,148.839
C03466=1141.353,305.996,-74.797,-176.954,8.694,148.839
C03467=1141.348,306.244,-74.829,-176.952,8.697,148.839
C03468=1141.344,306.493,-74.860,-176.949,8.701,148.839
C03469=1141.340,306.740,-74.891,-176.946,8.704,148.839
C03470=1141.336,306.988,-74.923,-176.944,8.707,148.839
C03471=1141.332,307.237,-74.954,-176.941,8.711,148.840
C03472=1141.328,307.484,-74.986,-176.938,8.714,148.840
C03473=1141.324,307.732,-75.018,-176.935,8.718,148.840
C03474=1141.319,307.980,-75.049,-176.933,8.721,148.840
C03475=1141.315,308.229,-75.081,-176.930,8.725,148.840
C03476=1141.311,308.477,-75.113,-176.927,8.729,148.840
C03477=1141.307,308.724,-75.144,-176.925,8.732,148.841
C03478=1141.303,308.972,-75.176,-176.922,8.736,148.841
C03479=1141.299,309.220,-75.207,-176.919,8.739,148.841
C03480=1141.294,309.468,-75.239,-176.917,8.742,148.841
C03481=1141.291,309.716,-75.271,-176.914,8.746,148.841
C03482=1141.286,309.964,-75.302,-176.912,8.750,148.841
C03483=1141.283,310.212,-75.334,-176.909,8.754,148.842
C03484=1141.278,310.460,-75.367,-176.906,8.757,148.842
C03485=1141.274,310.707,-75.398,-176.904,8.760,148.842
C03486=1141.270,310.956,-75.429,-176.901,8.764,148.842
C03487=1141.266,311.204,-75.461,-176.898,8.767,148.842
C03488=1141.261,311.452,-75.493,-176.895,8.771,148.842
C03489=1141.257,311.700,-75.525,-176.893,8.775,148.842
C03490=1141.254,311.948,-75.557,-176.890,8.779,148.843
C03491=1141.249,312.195,-75.589,-176.888,8.782,148.843
C03492=1141.245,312.443,-75.621,-176.885,8.785,148.843
C03493=1141.241,312.691,-75.653,-176.882,8.789,148.843
C03494=1141.236,312.969,-75.689,-176.879,8.793,148.843
C03495=1141.232,313.247,-75.725,-176.876,8.797,148.844
C03496=1141.227,313.525,-75.761,-176.873,8.801,148.844
C03497=1141.223,313.802,-75.796,-176.870,8.805,148.844
C03498=1141.219,314.050,-75.828,-176.868,8.808,148.844
C03499=1141.214,314.299,-75.861,-176.865,8.813,148.844
C03500=1141.211,314.547,-75.892,-176.863,8.816,148.845
C03501=1141.206,314.794,-75.925,-176.861,8.819,148.845
C03502=1141.202,315.042,-75.956,-176.857,8.823,148.845
C03503=1141.199,315.290,-75.989,-176.855,8.826,148.845
C03504=1141.194,315.538,-76.021,-176.852,8.830,148.845
C03505=1141.190,315.785,-76.053,-176.850,8.833,148.845
C03506=1141.185,316.034,-76.085,-176.847,8.837,148.846
C03507=1141.182,316.282,-76.117,-176.844,8.841,148.846
C03508=1141.178,316.530,-76.150,-176.841,8.845,148.846
C03509=1141.173,316.777,-76.182,-176.839,8.848,148.846
C03510=1141.169,317.025,-76.214,-176.837,8.851,148.846
C03511=1141.165,317.273,-76.247,-176.834,8.855,148.847
C03512=1141.161,317.521,-76.279,-176.831,8.859,148.847
C03513=1141.157,317.769,-76.311,-176.829,8.863,148.847
C03514=1141.153,318.017,-76.344,-176.826,8.866,148.847
C03515=1141.149,318.264,-76.376,-176.823,8.870,148.847
C03516=1141.144,318.512,-76.408,-176.821,8.873,148.848
C03517=1141.141,318.760,-76.441,-176.818,8.877,148.848
C03518=1141.136,319.008,-76.473,-176.816,8.881,148.848
C03519=1141.133,319.256,-76.505,-176.813,8.885,148.848
C03520=1141.129,319.504,-76.538,-176.810,8.888,148.848
C03521=1141.124,319.751,-76.570,-176.807,8.892,148.849
C03522=1141.120,319.999,-76.603,-176.805,8.895,148.849
C03523=1141.116,320.247,-76.635,-176.802,8.899,148.849
C03524=1141.112,320.495,-76.668,-176.800,8.903,148.849
C03525=1141.108,320.743,-76.700,-176.798,8.906,148.849
C03526=1141.104,320.991,-76.733,-176.795,8.910,148.850
C03527=1141.100,321.239,-76.765,-176.792,8.913,148.850
C03528=1141.096,321.487,-76.798,-176.789,8.917,148.850
C03529=1141.092,321.735,-76.830,-176.787,8.921,148.850
C03530=1141.088,321.982,-76.863,-176.784,8.925,148.851
C03531=1141.083,322.230,-76.895,-176.782,8.928,148.851
C03532=1141.080,322.478,-76.928,-176.779,8.932,148.851
C03533=1141.075,322.725,-76.961,-176.776,8.935,148.851
C03534=1141.071,322.974,-76.994,-176.774,8.939,148.851
C03535=1141.068,323.221,-77.026,-176.771,8.943,148.852
C03536=1141.063,323.469,-77.059,-176.768,8.947,148.852
C03537=1141.059,323.717,-77.092,-176.766,8.950,148.852
C03538=1141.055,323.965,-77.125,-176.763,8.954,148.852
C03539=1141.052,324.212,-77.157,-176.761,8.957,148.852
C03540=1141.047,324.461,-77.190,-176.758,8.962,148.853
C03541=1141.043,324.708,-77.223,-176.756,8.965,148.853
C03542=1141.039,324.956,-77.256,-176.753,8.969,148.853
C03543=1141.035,325.203,-77.289,-176.751,8.972,148.853
C03544=1141.031,325.452,-77.321,-176.748,8.976,148.854
C03545=1141.027,325.700,-77.354,-176.745,8.980,148.854
C03546=1141.023,325.947,-77.388,-176.742,8.984,148.854
C03547=1141.019,326.195,-77.421,-176.740,8.987,148.854
C03548=1141.015,326.442,-77.453,-176.737,8.991,148.854
C03549=1141.011,326.691,-77.486,-176.734,8.995,148.855
C03550=1141.007,326.939,-77.519,-176.732,8.999,148.855
C03551=1141.002,327.186,-77.552,-176.729,9.003,148.855
C03552=1140.998,327.434,-77.585,-176.727,9.006,148.856
C03553=1140.994,327.682,-77.618,-176.724,9.010,148.856
C03554=1140.990,327.929,-77.651,-176.722,9.013,148.856
C03555=1140.986,328.177,-77.685,-176.719,9.017,148.856
C03556=1140.982,328.425,-77.717,-176.716,9.021,148.856
C03557=1140.978,328.672,-77.750,-176.714,9.025,148.857
C03558=1140.974,328.920,-77.784,-176.712,9.028,148.857
C03559=1140.970,329.168,-77.817,-176.709,9.032,148.857
C03560=1140.967,329.416,-77.850,-176.706,9.036,148.857
C03561=1140.962,329.664,-77.883,-176.703,9.040,148.858
C03562=1140.958,329.912,-77.916,-176.701,9.043,148.858
C03563=1140.954,330.159,-77.950,-176.699,9.047,148.858
C03564=1140.950,330.407,-77.983,-176.696,9.051,148.859
C03565=1140.946,330.655,-78.016,-176.693,9.055,148.859
C03566=1140.942,330.903,-78.049,-176.690,9.059,148.859
C03567=1140.938,331.150,-78.082,-176.688,9.062,148.859
C03568=1140.933,331.398,-78.115,-176.685,9.066,148.859
C03569=1140.929,331.646,-78.149,-176.683,9.070,148.860
C03570=1140.926,331.894,-78.183,-176.680,9.074,148.860
C03571=1140.922,332.141,-78.216,-176.678,9.077,148.860
C03572=1140.918,332.389,-78.249,-176.675,9.081,148.860
C03573=1140.914,332.637,-78.282,-176.673,9.085,148.861
C03574=1140.909,332.884,-78.315,-176.670,9.089,148.861
C03575=1140.905,333.132,-78.349,-176.667,9.093,148.861
C03576=1140.901,333.380,-78.383,-176.665,9.096,148.862
C03577=1140.897,333.628,-78.417,-176.662,9.100,148.862
C03578=1140.893,333.876,-78.450,-176.660,9.104,148.862
C03579=1140.889,334.123,-78.484,-176.657,9.108,148.862
C03580=1140.885,334.371,-78.517,-176.654,9.112,148.863
C03581=1140.881,334.618,-78.550,-176.652,9.115,148.863
C03582=1140.878,334.866,-78.584,-176.649,9.120,148.863
C03583=1140.874,335.114,-78.617,-176.647,9.123,148.863
C03584=1140.869,335.362,-78.651,-176.644,9.127,148.864
C03585=1140.865,335.609,-78.685,-176.642,9.131,148.864
C03586=1140.861,335.857,-78.718,-176.639,9.134,148.864
C03587=1140.857,336.105,-78.752,-176.636,9.139,148.865
C03588=1140.853,336.352,-78.785,-176.634,9.142,148.865
C03589=1140.849,336.600,-78.819,-176.632,9.146,148.865
C03590=1140.845,336.847,-78.853,-176.629,9.149,148.865
C03591=1140.841,337.096,-78.887,-176.626,9.154,148.866
C03592=1140.837,337.343,-78.921,-176.624,9.158,148.866
C03593=1140.833,337.591,-78.954,-176.621,9.161,148.866
C03594=1140.829,337.839,-78.989,-176.619,9.165,148.867
C03595=1140.825,338.087,-79.022,-176.616,9.169,148.867
C03596=1140.821,338.334,-79.056,-176.614,9.173,148.867
C03597=1140.817,338.581,-79.089,-176.611,9.177,148.867
C03598=1140.812,338.862,-79.127,-176.608,9.181,148.868
C03599=1140.808,339.143,-79.166,-176.605,9.185,148.868
C03600=1140.804,339.424,-79.205,-176.602,9.190,148.868
C03601=1140.799,339.705,-79.243,-176.599,9.195,148.869
C03602=1140.795,339.952,-79.277,-176.597,9.198,148.869
C03603=1140.791,340.199,-79.310,-176.594,9.202,148.869
C03604=1140.787,340.448,-79.345,-176.592,9.206,148.870
C03605=1140.783,340.695,-79.379,-176.589,9.210,148.870
C03606=1140.779,340.942,-79.412,-176.586,9.214,148.870
C03607=1140.775,341.191,-79.447,-176.584,9.217,148.871
C03608=1140.771,341.438,-79.481,-176.581,9.221,148.871
C03609=1140.766,341.685,-79.515,-176.579,9.226,148.871
C03610=1140.763,341.933,-79.549,-176.577,9.229,148.872
C03611=1140.758,342.181,-79.583,-176.574,9.233,148.872
C03612=1140.755,342.428,-79.617,-176.572,9.237,148.872
C03613=1140.751,342.676,-79.651,-176.569,9.241,148.872
C03614=1140.747,342.923,-79.686,-176.566,9.245,148.873
C03615=1140.743,343.171,-79.719,-176.564,9.248,148.873
C03616=1140.739,343.419,-79.754,-176.561,9.253,148.873
C03617=1140.735,343.666,-79.787,-176.559,9.257,148.874
C03618=1140.731,343.914,-79.822,-176.556,9.260,148.874
C03619=1140.727,344.161,-79.856,-176.554,9.265,148.874
C03620=1140.722,344.409,-79.891,-176.551,9.269,148.875
C03621=1140.719,344.657,-79.925,-176.548,9.272,148.875
C03622=1140.715,344.904,-79.959,-176.546,9.276,148.875
C03623=1140.711,345.152,-79.994,-176.543,9.280,148.876
C03624=1140.707,345.399,-80.028,-176.541,9.284,148.876
C03625=1140.702,345.647,-80.062,-176.538,9.288,148.876
C03626=1140.699,345.895,-80.096,-176.536,9.292,148.877
C03627=1140.694,346.142,-80.131,-176.533,9.296,148.877
C03628=1140.691,346.390,-80.165,-176.531,9.300,148.877
C03629=1140.687,346.637,-80.200,-176.528,9.304,148.878
C03630=1140.683,346.885,-80.234,-176.526,9.307,148.878
C03631=1140.679,347.132,-80.269,-176.523,9.312,148.878
C03632=1140.675,347.381,-80.303,-176.520,9.316,148.878
C03633=1140.671,347.628,-80.337,-176.518,9.319,148.879
C03634=1140.667,347.876,-80.372,-176.515,9.324,148.879
C03635=1140.663,348.123,-80.407,-176.513,9.328,148.880
C03636=1140.659,348.371,-80.441,-176.510,9.331,148.880
C03637=1140.655,348.618,-80.475,-176.508,9.336,148.880
C03638=1140.651,348.866,-80.511,-176.505,9.340,148.880
C03639=1140.647,349.113,-80.545,-176.503,9.343,148.881
C03640=1140.643,349.361,-80.580,-176.500,9.347,148.881
C03641=1140.639,349.609,-80.614,-176.498,9.352,148.882
C03642=1140.635,349.856,-80.648,-176.495,9.355,148.882
C03643=1140.631,350.103,-80.683,-176.493,9.359,148.882
C03644=1140.627,350.351,-80.718,-176.490,9.363,148.882
C03645=1140.623,350.598,-80.752,-176.488,9.367,148.883
C03646=1140.620,350.846,-80.788,-176.485,9.371,148.883
C03647=1140.616,351.094,-80.823,-176.483,9.375,148.884
C03648=1140.611,351.341,-80.857,-176.481,9.379,148.884
C03649=1140.608,351.589,-80.892,-176.478,9.383,148.884
C03650=1140.604,351.836,-80.926,-176.475,9.387,148.885
C03651=1140.600,352.084,-80.961,-176.472,9.392,148.885
C03652=1140.595,352.331,-80.996,-176.470,9.395,148.885
C03653=1140.592,352.579,-81.031,-176.467,9.399,148.886
C03654=1140.588,352.827,-81.066,-176.465,9.404,148.886
C03655=1140.584,353.074,-81.101,-176.463,9.407,148.886
C03656=1140.580,353.322,-81.136,-176.460,9.411,148.887
C03657=1140.576,353.569,-81.171,-176.458,9.416,148.887
C03658=1140.572,353.817,-81.206,-176.455,9.420,148.887
C03659=1140.568,354.064,-81.241,-176.453,9.423,148.888
C03660=1140.564,354.311,-81.275,-176.450,9.427,148.888
C03661=1140.561,354.559,-81.311,-176.447,9.432,148.889
C03662=1140.557,354.807,-81.345,-176.445,9.435,148.889
C03663=1140.552,355.054,-81.381,-176.442,9.439,148.889
